# B&R Automation Studio project TrakDemo
Automation Studio 6.0.2.177; technology packages: mappCockpit 6.0.0, mappMotion 6.0.0, mappView 6.0.0, OpcUaCs 6.0.0

## Configuration Config1

CPU 5PC900.TS17-00, AutomationRuntime 6.0.2, Build 11.3.0, Safety 0.0, Vc 

### Task classes (Cpu.sw)
```
Cyclic#1:
  TrakInit <- Trak.TrakInit.prg
Cyclic#2:
  AssCtrl1 <- Trak.AssCtrl1.prg
  AssCtrl2 <- Trak.AssCtrl2.prg
DataObjects: McAcpSys
NcDataObjects: mcdrivelog
Binaries: FWRules, McAcpSim, arcoal, arsvcreg, TCData, McAcpDrv, mCoWebSc, mvLoader, arflatprv, udbdef, iomap, Config_1, arconfig, asfw, ashwac, sysconf, User, Settings, Role, ashwd, Config_4, Config_3, Config_2, Config, Hierarchy
Libraries: McBase, CoTrace, AsZip, FileIO, runtime, McAxis, McAcpTrak, MpBase, TrakLib, standard, AsBrStr, sys_lib, brsystem, TrakDiag, astime, ArEventLog, DataObj, AsHttp, AsArSdm, MpAxis, McAcpAx, powerlnk, arssl, asieccon, asepl
```

### Hardware
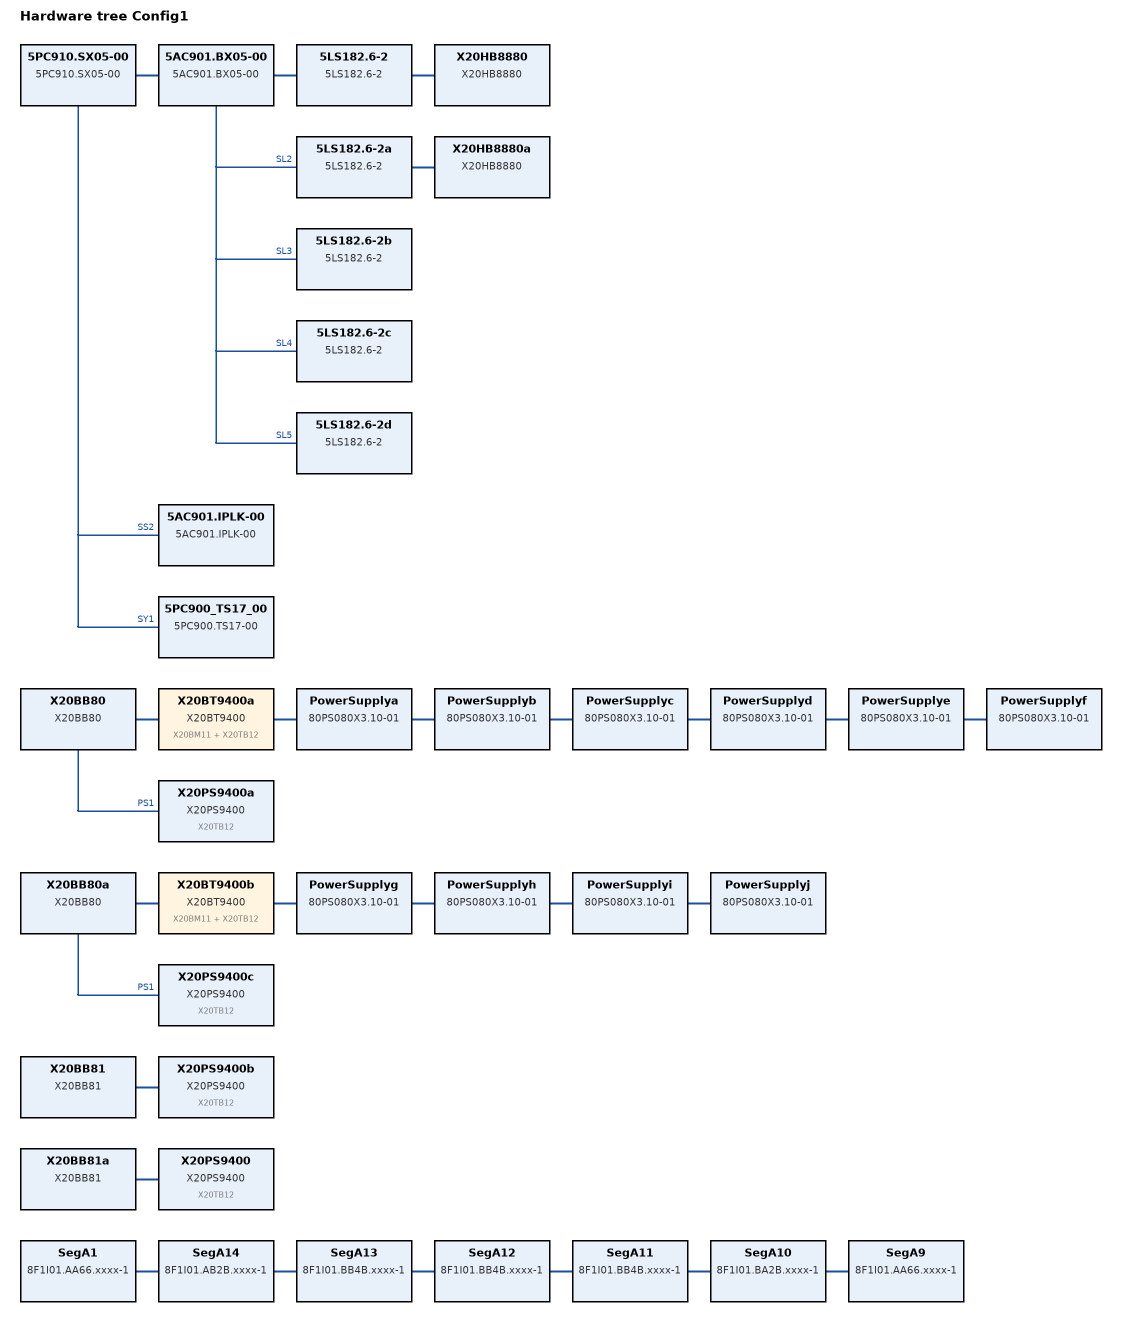
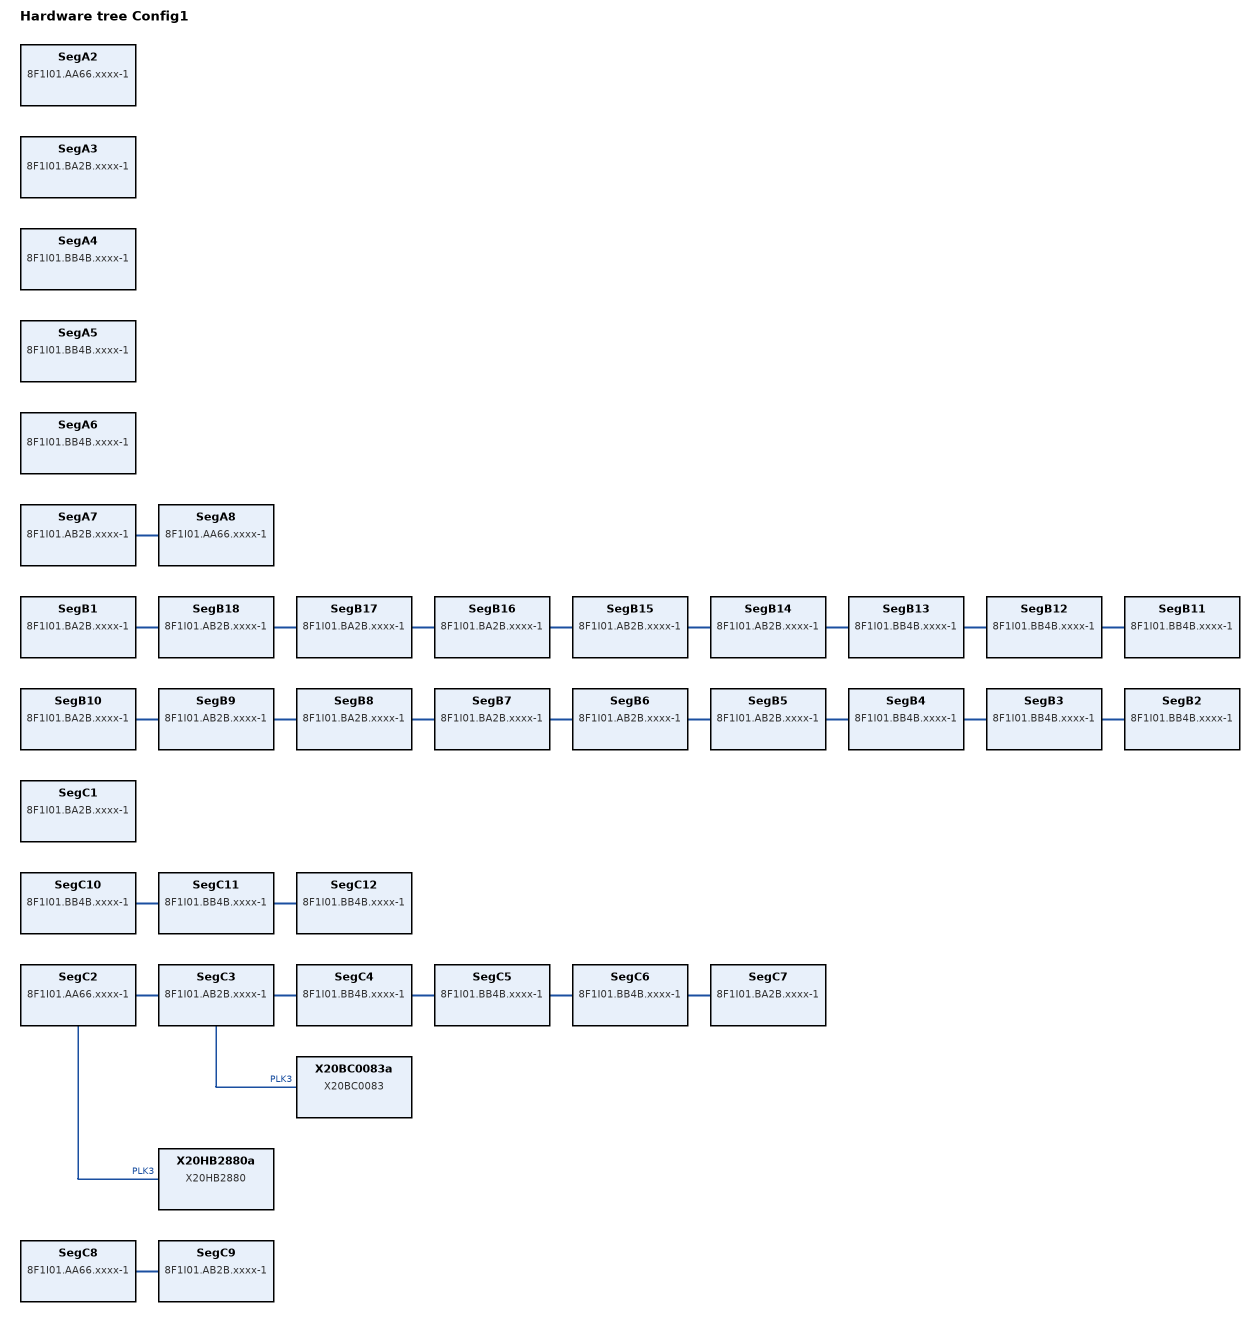
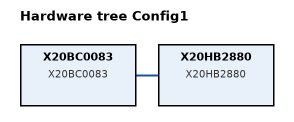
```
5AC901.BX05-00 : 5AC901.BX05-00 v1.0.1.0  [SY -> 5PC910.SX05-00.SY3]
5AC901.IPLK-00 : 5AC901.IPLK-00 v2.0.0.0 (Disabled=true)  [SS -> 5PC910.SX05-00.SS2]
  Connector IF1 (Disabled=true)
5LS182.6-2 : 5LS182.6-2 v1.12.0.0  [SL -> 5AC901.BX05-00.SL1]
  Connector IF1:
    NodeDefinition = Software
5LS182.6-2a : 5LS182.6-2 v1.12.0.0  [SL -> 5AC901.BX05-00.SL2]
5LS182.6-2b : 5LS182.6-2 v1.12.0.0 (Disabled=true)  [SL -> 5AC901.BX05-00.SL3]
  Connector IF1 (Disabled=true)
5LS182.6-2c : 5LS182.6-2 v1.12.0.0 (Disabled=true)  [SL -> 5AC901.BX05-00.SL4]
  Connector IF1 (Disabled=true)
5LS182.6-2d : 5LS182.6-2 v1.12.0.0 (Disabled=true)  [SL -> 5AC901.BX05-00.SL5]
  Connector IF1 (Disabled=true)
5PC900_TS17_00 : 5PC900.TS17-00 v2.1.0.0  [SY -> 5PC910.SX05-00.SY1]
  ConfigurationID = TrakDemo_Config1
  ConfigVersion = 1.2.3
  MotionLoggerSize = 2048000
  SystemTick = 2000
  TaskClassIdleTime = 10000
  Cyclic1Tolerance = 0
  FileDevice1
  FileDeviceName1 = SvgData
  FileDevicePath1 = USER_PATH\web\SvgData
  FileDevice2
  FileDeviceName2 = Diagnosis
  FileDevicePath2 = USER_PATH\web\Diagnosis
  EthernetDefaultGateway = 10.24.153.1
  ActivateFtpServer = 1
  FtpUser1
  FtpUsername1 = bur
  FtpUserPassword1 = efcpoAfz3gk2rn0a9Nq2v7CfehAGIZc7rIbAOhV34KU=
  FtpUserSalt1 = 5Q6RY3ay
  FTPAccessRight1 = 0
  ActivateWebServer = 1
  WebServerProtocol = 1
  WebServerWebDir = F:\web\
  ActivateSdm = 1
5PC910.SX05-00 : 5PC910.SX05-00 v2.1.2.0
  Connector IF1:
    AssignedOperatingSystem = ARemb
  Connector IF3:
    AssignedOperatingSystem = ARemb
    ActivateDevice = 1
    Mode = Manual
    InternetAddress = 10.24.153.43
    SubnetMask = 255.255.255.192
    ActivateIna = 0
    ActivateSnmp = 2
  Connector IF4:
    AssignedOperatingSystem = ARemb
    ActivateDevice = 1
  Connector IF5:
    AssignedOperatingSystem = ARemb
  Connector IF6:
    AssignedOperatingSystem = ARemb
  Connector IF7:
    AssignedOperatingSystem = ARemb
  Connector IF8:
    AssignedOperatingSystem = ARemb
  Connector IF9:
    AssignedOperatingSystem = ARemb
PowerSupplya : 80PS080X3.10-01 v1.7.0.0  [X2X1 -> X20BT9400a.X2X1 [Cable Type=X2XCable, Length=10, Version=1.0.0.3]]
  Supervision = off
PowerSupplyb : 80PS080X3.10-01 v1.7.0.0  [X2X1 -> PowerSupplya.X2X2 [Cable Type=X2XCable, Length=10, Version=1.0.0.3]]
  Supervision = off
PowerSupplyc : 80PS080X3.10-01 v1.7.0.0  [X2X1 -> PowerSupplyb.X2X2 [Cable Type=X2XCable, Length=10, Version=1.0.0.3]]
  Supervision = off
PowerSupplyd : 80PS080X3.10-01 v1.7.0.0  [X2X1 -> PowerSupplyc.X2X2 [Cable Type=X2XCable, Length=10, Version=1.0.0.3]]
  Supervision = off
PowerSupplye : 80PS080X3.10-01 v1.7.0.0  [X2X1 -> PowerSupplyd.X2X2 [Cable Type=X2XCable, Length=10, Version=1.0.0.3]]
  Supervision = off
PowerSupplyf : 80PS080X3.10-01 v1.7.0.0  [X2X1 -> PowerSupplye.X2X2 [Cable Type=X2XCable, Length=10, Version=1.0.0.3]]
  Supervision = off
PowerSupplyg : 80PS080X3.10-01 v1.7.0.0  [X2X1 -> X20BT9400b.X2X1 [Cable Type=X2XCable, Length=10, Version=1.0.0.3]]
  Supervision = off
PowerSupplyh : 80PS080X3.10-01 v1.7.0.0  [X2X1 -> PowerSupplyg.X2X2 [Cable Type=X2XCable, Length=10, Version=1.0.0.3]]
  Supervision = off
PowerSupplyi : 80PS080X3.10-01 v1.7.0.0  [X2X1 -> PowerSupplyh.X2X2 [Cable Type=X2XCable, Length=10, Version=1.0.0.3]]
  Supervision = off
PowerSupplyj : 80PS080X3.10-01 v1.7.0.0  [X2X1 -> PowerSupplyi.X2X2 [Cable Type=X2XCable, Length=10, Version=1.0.0.3]]
  Supervision = off
SegA1 : 8F1I01.AA66.xxxx-1 v1.0.0.4 (NodeNumber=1)  [PLK1 -> SegA2.PLK2 [Cable Type=PowerlinkCable, Length=10, Version=1.0.0.3]; PLK2 -> SegA14.PLK1 [Cable Type=PowerlinkCable, Length=10, Version=1.0.0.3]; PLK3 -> X20HB8880.ETH2 [Cable Type=PowerlinkCable, Length=10, Version=1.0.0.3]]
  DriveConfiguration:
    McTypeID = LLMConfig
  DriveConfiguration/Segment:
    Shape = STRAIGHT660
    SegmentReference = gSegA1
    SegmentSectorDirection = Positive
    ElongationCompensation = UseAssemblySetting
    StopReaction = UseAssemblySetting
    SpeedFilter = UseAssemblySetting
SegA10 : 8F1I01.BA2B.xxxx-1 v1.0.0.4 (NodeNumber=25)  [PLK1 -> SegA11.PLK2 [Cable Type=PowerlinkCable, Length=10, Version=1.0.0.3]; PLK2 -> SegA9.PLK1 [Cable Type=PowerlinkCable, Length=10, Version=1.0.0.3]]
  DriveConfiguration:
    McTypeID = LLMConfig
  DriveConfiguration/Segment:
    Shape = CIRCULAR_TO_STRAIGHT105
    SegmentReference = gSegA10
    SegmentSectorDirection = Positive
    ElongationCompensation = UseAssemblySetting
    StopReaction = UseAssemblySetting
    SpeedFilter = UseAssemblySetting
SegA11 : 8F1I01.BB4B.xxxx-1 v1.0.0.4 (NodeNumber=24)  [PLK1 -> SegA12.PLK2 [Cable Type=PowerlinkCable, Length=10, Version=1.0.0.3]; PLK2 -> SegA10.PLK1 [Cable Type=PowerlinkCable, Length=10, Version=1.0.0.3]]
  DriveConfiguration:
    McTypeID = LLMConfig
  DriveConfiguration/Segment:
    Shape = CIRCULAR
    SegmentReference = gSegA11
    SegmentSectorDirection = Positive
    ElongationCompensation = UseAssemblySetting
    StopReaction = UseAssemblySetting
    SpeedFilter = UseAssemblySetting
SegA12 : 8F1I01.BB4B.xxxx-1 v1.0.0.4 (NodeNumber=23)  [PLK1 -> SegA13.PLK2 [Cable Type=PowerlinkCable, Length=10, Version=1.0.0.3]; PLK2 -> SegA11.PLK1 [Cable Type=PowerlinkCable, Length=10, Version=1.0.0.3]]
  DriveConfiguration:
    McTypeID = LLMConfig
  DriveConfiguration/Segment:
    Shape = CIRCULAR
    SegmentReference = gSegA12
    SegmentSectorDirection = Positive
    ElongationCompensation = UseAssemblySetting
    StopReaction = UseAssemblySetting
    SpeedFilter = UseAssemblySetting
SegA13 : 8F1I01.BB4B.xxxx-1 v1.0.0.4 (NodeNumber=22)  [PLK1 -> SegA14.PLK2 [Cable Type=PowerlinkCable, Length=10, Version=1.0.0.3]; PLK2 -> SegA12.PLK1 [Cable Type=PowerlinkCable, Length=10, Version=1.0.0.3]]
  DriveConfiguration:
    McTypeID = LLMConfig
  DriveConfiguration/Segment:
    Shape = CIRCULAR
    SegmentReference = gSegA13
    SegmentSectorDirection = Positive
    ElongationCompensation = UseAssemblySetting
    StopReaction = UseAssemblySetting
    SpeedFilter = UseAssemblySetting
SegA14 : 8F1I01.AB2B.xxxx-1 v1.0.0.4 (NodeNumber=21)  [PLK1 -> SegA1.PLK2 [Cable Type=PowerlinkCable, Length=10, Version=1.0.0.3]; PLK2 -> SegA13.PLK1 [Cable Type=PowerlinkCable, Length=10, Version=1.0.0.3]]
  DriveConfiguration:
    McTypeID = LLMConfig
  DriveConfiguration/Segment:
    Shape = STRAIGHT105_TO_CIRCULAR
    SegmentReference = gSegA14
    SegmentSectorDirection = Positive
    ElongationCompensation = UseAssemblySetting
    StopReaction = UseAssemblySetting
    SpeedFilter = UseAssemblySetting
SegA2 : 8F1I01.AA66.xxxx-1 v1.0.0.4 (NodeNumber=2)  [PLK1 -> SegA3.PLK2 [Cable Type=PowerlinkCable, Length=10, Version=1.0.0.3]; PLK2 -> SegA1.PLK1 [Cable Type=PowerlinkCable, Length=10, Version=1.0.0.3]]
  DriveConfiguration:
    McTypeID = LLMConfig
  DriveConfiguration/Segment:
    Shape = STRAIGHT660
    SegmentReference = gSegA2
    SegmentSectorDirection = Positive
    ElongationCompensation = UseAssemblySetting
    StopReaction = UseAssemblySetting
    SpeedFilter = UseAssemblySetting
SegA3 : 8F1I01.BA2B.xxxx-1 v1.0.0.4 (NodeNumber=27)  [PLK1 -> SegA4.PLK2 [Cable Type=PowerlinkCable, Length=10, Version=1.0.0.3]; PLK2 -> SegA2.PLK1 [Cable Type=PowerlinkCable, Length=10, Version=1.0.0.3]]
  DriveConfiguration:
    McTypeID = LLMConfig
  DriveConfiguration/Segment:
    Shape = CIRCULAR_TO_STRAIGHT105
    SegmentReference = gSegA3
    SegmentSectorDirection = Positive
    ElongationCompensation = UseAssemblySetting
    StopReaction = UseAssemblySetting
    SpeedFilter = UseAssemblySetting
SegA4 : 8F1I01.BB4B.xxxx-1 v1.0.0.4 (NodeNumber=28)  [PLK1 -> SegA5.PLK2 [Cable Type=PowerlinkCable, Length=10, Version=1.0.0.3]; PLK2 -> SegA3.PLK1 [Cable Type=PowerlinkCable, Length=10, Version=1.0.0.3]]
  DriveConfiguration:
    McTypeID = LLMConfig
  DriveConfiguration/Segment:
    Shape = CIRCULAR
    SegmentReference = gSegA4
    SegmentSectorDirection = Positive
    ElongationCompensation = UseAssemblySetting
    StopReaction = UseAssemblySetting
    SpeedFilter = UseAssemblySetting
SegA5 : 8F1I01.BB4B.xxxx-1 v1.0.0.4 (NodeNumber=29)  [PLK1 -> SegA6.PLK2 [Cable Type=PowerlinkCable, Length=10, Version=1.0.0.3]; PLK2 -> SegA4.PLK1 [Cable Type=PowerlinkCable, Length=10, Version=1.0.0.3]]
  DriveConfiguration:
    McTypeID = LLMConfig
  DriveConfiguration/Segment:
    Shape = CIRCULAR
    SegmentReference = gSegA5
    SegmentSectorDirection = Positive
    ElongationCompensation = UseAssemblySetting
    StopReaction = UseAssemblySetting
    SpeedFilter = UseAssemblySetting
SegA6 : 8F1I01.BB4B.xxxx-1 v1.0.0.4 (NodeNumber=30)  [PLK1 -> SegA7.PLK2 [Cable Type=PowerlinkCable, Length=10, Version=1.0.0.3]; PLK2 -> SegA5.PLK1 [Cable Type=PowerlinkCable, Length=10, Version=1.0.0.3]]
  DriveConfiguration:
    McTypeID = LLMConfig
  DriveConfiguration/Segment:
    Shape = CIRCULAR
    SegmentReference = gSegA6
    SegmentSectorDirection = Positive
    ElongationCompensation = UseAssemblySetting
    StopReaction = UseAssemblySetting
    SpeedFilter = UseAssemblySetting
SegA7 : 8F1I01.AB2B.xxxx-1 v1.0.0.4 (NodeNumber=31)  [PLK1 -> SegA8.PLK2 [Cable Type=PowerlinkCable, Length=10, Version=1.0.0.3]; PLK2 -> SegA6.PLK1 [Cable Type=PowerlinkCable, Length=10, Version=1.0.0.3]]
  DriveConfiguration:
    McTypeID = LLMConfig
  DriveConfiguration/Segment:
    Shape = STRAIGHT105_TO_CIRCULAR
    SegmentReference = gSegA7
    SegmentSectorDirection = Positive
    ElongationCompensation = UseAssemblySetting
    StopReaction = UseAssemblySetting
    SpeedFilter = UseAssemblySetting
SegA8 : 8F1I01.AA66.xxxx-1 v1.0.0.4 (NodeNumber=32)  [PLK2 -> SegA7.PLK1 [Cable Type=PowerlinkCable, Length=10, Version=1.0.0.3]]
  DriveConfiguration:
    McTypeID = LLMConfig
  DriveConfiguration/Segment:
    Shape = STRAIGHT660
    SegmentReference = gSegA8
    SegmentSectorDirection = Positive
    ElongationCompensation = UseAssemblySetting
    StopReaction = UseAssemblySetting
    SpeedFilter = UseAssemblySetting
SegA9 : 8F1I01.AA66.xxxx-1 v1.0.0.4 (NodeNumber=26)  [PLK1 -> SegA10.PLK2 [Cable Type=PowerlinkCable, Length=10, Version=1.0.0.3]]
  DriveConfiguration:
    McTypeID = LLMConfig
  DriveConfiguration/Segment:
    Shape = STRAIGHT660
    SegmentReference = gSegA9
    SegmentSectorDirection = Positive
    ElongationCompensation = UseAssemblySetting
    StopReaction = UseAssemblySetting
    SpeedFilter = UseAssemblySetting
SegB1 : 8F1I01.BA2B.xxxx-1 v1.0.0.4 (NodeNumber=3)  [PLK1 -> SegB2.PLK2 [Cable Type=PowerlinkCable, Length=10, Version=1.0.0.3]; PLK2 -> SegB18.PLK1 [Cable Type=PowerlinkCable, Length=10, Version=1.0.0.3]; PLK3 -> X20HB2880.ETH2 [Cable Type=PowerlinkCable, Length=10, Version=1.0.0.3]]
  DriveConfiguration:
    McTypeID = LLMConfig
  DriveConfiguration/Segment:
    Shape = CIRCULAR_TO_STRAIGHT105
    SegmentReference = gSegB1
    SegmentSectorDirection = Positive
    ElongationCompensation = UseAssemblySetting
    StopReaction = UseAssemblySetting
    SpeedFilter = UseAssemblySetting
SegB10 : 8F1I01.BA2B.xxxx-1 v1.0.0.4 (NodeNumber=12)  [PLK2 -> SegB9.PLK1 [Cable Type=PowerlinkCable, Length=10, Version=1.0.0.3]]
  DriveConfiguration:
    McTypeID = LLMConfig
  DriveConfiguration/Segment:
    Shape = CIRCULAR_TO_STRAIGHT105
    SegmentReference = gSegB10
    SegmentSectorDirection = Positive
    ElongationCompensation = UseAssemblySetting
    StopReaction = UseAssemblySetting
    SpeedFilter = UseAssemblySetting
SegB11 : 8F1I01.BB4B.xxxx-1 v1.0.0.4 (NodeNumber=11)  [PLK1 -> SegB12.PLK2 [Cable Type=PowerlinkCable, Length=10, Version=1.0.0.3]]
  DriveConfiguration:
    McTypeID = LLMConfig
  DriveConfiguration/Segment:
    Shape = CIRCULAR
    SegmentReference = gSegB11
    SegmentSectorDirection = Positive
    ElongationCompensation = UseAssemblySetting
    StopReaction = UseAssemblySetting
    SpeedFilter = UseAssemblySetting
SegB12 : 8F1I01.BB4B.xxxx-1 v1.0.0.4 (NodeNumber=10)  [PLK1 -> SegB13.PLK2 [Cable Type=PowerlinkCable, Length=10, Version=1.0.0.3]; PLK2 -> SegB11.PLK1 [Cable Type=PowerlinkCable, Length=10, Version=1.0.0.3]]
  DriveConfiguration:
    McTypeID = LLMConfig
  DriveConfiguration/Segment:
    Shape = CIRCULAR
    SegmentReference = gSegB12
    SegmentSectorDirection = Positive
    ElongationCompensation = UseAssemblySetting
    StopReaction = UseAssemblySetting
    SpeedFilter = UseAssemblySetting
SegB13 : 8F1I01.BB4B.xxxx-1 v1.0.0.4 (NodeNumber=9)  [PLK1 -> SegB14.PLK2 [Cable Type=PowerlinkCable, Length=10, Version=1.0.0.3]; PLK2 -> SegB12.PLK1 [Cable Type=PowerlinkCable, Length=10, Version=1.0.0.3]]
  DriveConfiguration:
    McTypeID = LLMConfig
  DriveConfiguration/Segment:
    Shape = CIRCULAR
    SegmentReference = gSegB13
    SegmentSectorDirection = Positive
    ElongationCompensation = UseAssemblySetting
    StopReaction = UseAssemblySetting
    SpeedFilter = UseAssemblySetting
SegB14 : 8F1I01.AB2B.xxxx-1 v1.0.0.4 (NodeNumber=8)  [PLK1 -> SegB15.PLK2 [Cable Type=PowerlinkCable, Length=10, Version=1.0.0.3]; PLK2 -> SegB13.PLK1 [Cable Type=PowerlinkCable, Length=10, Version=1.0.0.3]]
  DriveConfiguration:
    McTypeID = LLMConfig
  DriveConfiguration/Segment:
    Shape = STRAIGHT105_TO_CIRCULAR
    SegmentReference = gSegB14
    SegmentSectorDirection = Positive
    ElongationCompensation = UseAssemblySetting
    StopReaction = UseAssemblySetting
    SpeedFilter = UseAssemblySetting
SegB15 : 8F1I01.AB2B.xxxx-1 v1.0.0.4 (NodeNumber=7)  [PLK1 -> SegB16.PLK2 [Cable Type=PowerlinkCable, Length=10, Version=1.0.0.3]; PLK2 -> SegB14.PLK1 [Cable Type=PowerlinkCable, Length=10, Version=1.0.0.3]]
  DriveConfiguration:
    McTypeID = LLMConfig
  DriveConfiguration/Segment:
    Shape = STRAIGHT105_TO_CIRCULAR
    SegmentReference = gSegB15
    SegmentSectorDirection = Positive
    ElongationCompensation = UseAssemblySetting
    StopReaction = UseAssemblySetting
    SpeedFilter = UseAssemblySetting
SegB16 : 8F1I01.BA2B.xxxx-1 v1.0.0.4 (NodeNumber=6)  [PLK1 -> SegB17.PLK2 [Cable Type=PowerlinkCable, Length=10, Version=1.0.0.3]; PLK2 -> SegB15.PLK1 [Cable Type=PowerlinkCable, Length=10, Version=1.0.0.3]]
  DriveConfiguration:
    McTypeID = LLMConfig
  DriveConfiguration/Segment:
    Shape = CIRCULAR_TO_STRAIGHT105
    SegmentReference = gSegB16
    SegmentSectorDirection = Positive
    ElongationCompensation = UseAssemblySetting
    StopReaction = UseAssemblySetting
    SpeedFilter = UseAssemblySetting
SegB17 : 8F1I01.BA2B.xxxx-1 v1.0.0.4 (NodeNumber=5)  [PLK1 -> SegB18.PLK2 [Cable Type=PowerlinkCable, Length=10, Version=1.0.0.3]; PLK2 -> SegB16.PLK1 [Cable Type=PowerlinkCable, Length=10, Version=1.0.0.3]]
  DriveConfiguration:
    McTypeID = LLMConfig
  DriveConfiguration/Segment:
    Shape = CIRCULAR_TO_STRAIGHT105
    SegmentReference = gSegB17
    SegmentSectorDirection = Positive
    ElongationCompensation = UseAssemblySetting
    StopReaction = UseAssemblySetting
    SpeedFilter = UseAssemblySetting
SegB18 : 8F1I01.AB2B.xxxx-1 v1.0.0.4 (NodeNumber=4)  [PLK1 -> SegB1.PLK2 [Cable Type=PowerlinkCable, Length=10, Version=1.0.0.3]; PLK2 -> SegB17.PLK1 [Cable Type=PowerlinkCable, Length=10, Version=1.0.0.3]]
  DriveConfiguration:
    McTypeID = LLMConfig
  DriveConfiguration/Segment:
    Shape = STRAIGHT105_TO_CIRCULAR
    SegmentReference = gSegB18
    SegmentSectorDirection = Positive
    ElongationCompensation = UseAssemblySetting
    StopReaction = UseAssemblySetting
    SpeedFilter = UseAssemblySetting
SegB2 : 8F1I01.BB4B.xxxx-1 v1.0.0.4 (NodeNumber=13)  [PLK1 -> SegB3.PLK2 [Cable Type=PowerlinkCable, Length=10, Version=1.0.0.3]; PLK2 -> SegB1.PLK1 [Cable Type=PowerlinkCable, Length=10, Version=1.0.0.3]]
  DriveConfiguration:
    McTypeID = LLMConfig
  DriveConfiguration/Segment:
    Shape = CIRCULAR
    SegmentReference = gSegB2
    SegmentSectorDirection = Positive
    ElongationCompensation = UseAssemblySetting
    StopReaction = UseAssemblySetting
    SpeedFilter = UseAssemblySetting
SegB3 : 8F1I01.BB4B.xxxx-1 v1.0.0.4 (NodeNumber=14)  [PLK1 -> SegB4.PLK2 [Cable Type=PowerlinkCable, Length=10, Version=1.0.0.3]; PLK2 -> SegB2.PLK1 [Cable Type=PowerlinkCable, Length=10, Version=1.0.0.3]]
  DriveConfiguration:
    McTypeID = LLMConfig
  DriveConfiguration/Segment:
    Shape = CIRCULAR
    SegmentReference = gSegB3
    SegmentSectorDirection = Positive
    ElongationCompensation = UseAssemblySetting
    StopReaction = UseAssemblySetting
    SpeedFilter = UseAssemblySetting
SegB4 : 8F1I01.BB4B.xxxx-1 v1.0.0.4 (NodeNumber=15)  [PLK1 -> SegB5.PLK2 [Cable Type=PowerlinkCable, Length=10, Version=1.0.0.3]; PLK2 -> SegB3.PLK1 [Cable Type=PowerlinkCable, Length=10, Version=1.0.0.3]]
  DriveConfiguration:
    McTypeID = LLMConfig
  DriveConfiguration/Segment:
    Shape = CIRCULAR
    SegmentReference = gSegB4
    SegmentSectorDirection = Positive
    ElongationCompensation = UseAssemblySetting
    StopReaction = UseAssemblySetting
    SpeedFilter = UseAssemblySetting
SegB5 : 8F1I01.AB2B.xxxx-1 v1.0.0.4 (NodeNumber=16)  [PLK1 -> SegB6.PLK2 [Cable Type=PowerlinkCable, Length=10, Version=1.0.0.3]; PLK2 -> SegB4.PLK1 [Cable Type=PowerlinkCable, Length=10, Version=1.0.0.3]]
  DriveConfiguration:
    McTypeID = LLMConfig
  DriveConfiguration/Segment:
    Shape = STRAIGHT105_TO_CIRCULAR
    SegmentReference = gSegB5
    SegmentSectorDirection = Positive
    ElongationCompensation = UseAssemblySetting
    StopReaction = UseAssemblySetting
    SpeedFilter = UseAssemblySetting
SegB6 : 8F1I01.AB2B.xxxx-1 v1.0.0.4 (NodeNumber=17)  [PLK1 -> SegB7.PLK2 [Cable Type=PowerlinkCable, Length=10, Version=1.0.0.3]; PLK2 -> SegB5.PLK1 [Cable Type=PowerlinkCable, Length=10, Version=1.0.0.3]]
  DriveConfiguration:
    McTypeID = LLMConfig
  DriveConfiguration/Segment:
    Shape = STRAIGHT105_TO_CIRCULAR
    SegmentReference = gSegB6
    SegmentSectorDirection = Positive
    ElongationCompensation = UseAssemblySetting
    StopReaction = UseAssemblySetting
    SpeedFilter = UseAssemblySetting
SegB7 : 8F1I01.BA2B.xxxx-1 v1.0.0.4 (NodeNumber=18)  [PLK1 -> SegB8.PLK2 [Cable Type=PowerlinkCable, Length=10, Version=1.0.0.3]; PLK2 -> SegB6.PLK1 [Cable Type=PowerlinkCable, Length=10, Version=1.0.0.3]]
  DriveConfiguration:
    McTypeID = LLMConfig
  DriveConfiguration/Segment:
    Shape = CIRCULAR_TO_STRAIGHT105
    SegmentReference = gSegB7
    SegmentSectorReference = gSecB7
    SegmentSectorDirection = Positive
    ElongationCompensation = UseAssemblySetting
    ACC = Inactive
    StopReaction = UseAssemblySetting
    SpeedFilter = UseAssemblySetting
    PositionControllerLagMonitor = UseAssemblySetting
SegB8 : 8F1I01.BA2B.xxxx-1 v1.0.0.4 (NodeNumber=20)  [PLK1 -> SegB9.PLK2 [Cable Type=PowerlinkCable, Length=10, Version=1.0.0.3]; PLK2 -> SegB7.PLK1 [Cable Type=PowerlinkCable, Length=10, Version=1.0.0.3]]
  DriveConfiguration:
    McTypeID = LLMConfig
  DriveConfiguration/Segment:
    Shape = CIRCULAR_TO_STRAIGHT105
    SegmentReference = gSegB8
    SegmentSectorDirection = Positive
    ElongationCompensation = UseAssemblySetting
    StopReaction = UseAssemblySetting
    SpeedFilter = UseAssemblySetting
SegB9 : 8F1I01.AB2B.xxxx-1 v1.0.0.4 (NodeNumber=19)  [PLK1 -> SegB10.PLK2 [Cable Type=PowerlinkCable, Length=10, Version=1.0.0.3]; PLK2 -> SegB8.PLK1 [Cable Type=PowerlinkCable, Length=10, Version=1.0.0.3]]
  DriveConfiguration:
    McTypeID = LLMConfig
  DriveConfiguration/Segment:
    Shape = STRAIGHT105_TO_CIRCULAR
    SegmentReference = gSegB9
    SegmentSectorDirection = Positive
    ElongationCompensation = UseAssemblySetting
    StopReaction = UseAssemblySetting
    SpeedFilter = UseAssemblySetting
SegC1 : 8F1I01.BA2B.xxxx-1 v1.0.0.4 (NodeNumber=1)  [PLK1 -> SegC12.PLK2 [Cable Type=PowerlinkCable, Length=10, Version=1.0.0.3]; PLK3 -> X20HB8880a.ETH2 [Cable Type=PowerlinkCable, Length=10, Version=1.0.0.3]]
  DriveConfiguration:
    McTypeID = LLMConfig
  DriveConfiguration/Segment:
    Shape = CIRCULAR_TO_STRAIGHT105
    SegmentReference = gSegC1
    SegmentSectorReference = gSecC1
    SegmentSectorDirection = Positive
    ElongationCompensation = UseAssemblySetting
    ACC = Inactive
    StopReaction = UseAssemblySetting
    SpeedFilter = UseAssemblySetting
    PositionControllerLagMonitor = UseAssemblySetting
SegC10 : 8F1I01.BB4B.xxxx-1 v1.0.0.4  [PLK1 -> SegC9.PLK2 [Cable Type=PowerlinkCable, Length=10, Version=1.0.0.3]; PLK2 -> SegC11.PLK1 [Cable Type=PowerlinkCable, Length=10, Version=1.0.0.3]]
  DriveConfiguration:
    McTypeID = LLMConfig
  DriveConfiguration/Segment:
    Shape = CIRCULAR
    SegmentReference = gSegC10
    SegmentSectorDirection = Positive
    ElongationCompensation = UseAssemblySetting
    ACC = Inactive
    StopReaction = UseAssemblySetting
    SpeedFilter = UseAssemblySetting
    PositionControllerLagMonitor = UseAssemblySetting
SegC11 : 8F1I01.BB4B.xxxx-1 v1.0.0.4  [PLK1 -> SegC10.PLK2 [Cable Type=PowerlinkCable, Length=10, Version=1.0.0.3]; PLK2 -> SegC12.PLK1 [Cable Type=PowerlinkCable, Length=10, Version=1.0.0.3]]
  DriveConfiguration:
    McTypeID = LLMConfig
  DriveConfiguration/Segment:
    Shape = CIRCULAR
    SegmentReference = gSegC11
    SegmentSectorDirection = Positive
    ElongationCompensation = UseAssemblySetting
    ACC = Inactive
    StopReaction = UseAssemblySetting
    SpeedFilter = UseAssemblySetting
    PositionControllerLagMonitor = UseAssemblySetting
SegC12 : 8F1I01.BB4B.xxxx-1 v1.0.0.4 (NodeNumber=3)  [PLK1 -> SegC11.PLK2 [Cable Type=PowerlinkCable, Length=10, Version=1.0.0.3]; PLK2 -> SegC1.PLK1 [Cable Type=PowerlinkCable, Length=10, Version=1.0.0.3]]
  DriveConfiguration:
    McTypeID = LLMConfig
  DriveConfiguration/Segment:
    Shape = CIRCULAR
    SegmentReference = gSegC12
    SegmentSectorDirection = Positive
    ElongationCompensation = UseAssemblySetting
    ACC = Inactive
    StopReaction = UseAssemblySetting
    SpeedFilter = UseAssemblySetting
    PositionControllerLagMonitor = UseAssemblySetting
SegC2 : 8F1I01.AA66.xxxx-1 v1.0.0.4 (NodeNumber=2)  [PLK2 -> SegC3.PLK1 [Cable Type=PowerlinkCable, Length=10, Version=1.0.0.3]; PLK3 -> X20HB2880a.ETH2 [Cable Type=PowerlinkCable, Length=10, Version=1.0.0.3]]
  DriveConfiguration:
    McTypeID = LLMConfig
  DriveConfiguration/Segment:
    Shape = STRAIGHT660
    SegmentReference = gSegC2
    SegmentSectorDirection = Positive
    ElongationCompensation = UseAssemblySetting
    ACC = Inactive
    StopReaction = UseAssemblySetting
    SpeedFilter = UseAssemblySetting
    PositionControllerLagMonitor = UseAssemblySetting
SegC3 : 8F1I01.AB2B.xxxx-1 v1.0.0.4 (NodeNumber=12)  [PLK1 -> SegC2.PLK2 [Cable Type=PowerlinkCable, Length=10, Version=1.0.0.3]; PLK2 -> SegC4.PLK1 [Cable Type=PowerlinkCable, Length=10, Version=1.0.0.3]; PLK3 -> X20BC0083a.PLK1 [Cable Type=PowerlinkCable, Length=10, Version=1.0.0.3]]
  DriveConfiguration:
    McTypeID = LLMConfig
  DriveConfiguration/Segment:
    Shape = STRAIGHT105_TO_CIRCULAR
    SegmentReference = gSegC3
    SegmentSectorDirection = Positive
    ElongationCompensation = UseAssemblySetting
    ACC = Inactive
    StopReaction = UseAssemblySetting
    SpeedFilter = UseAssemblySetting
    PositionControllerLagMonitor = UseAssemblySetting
SegC4 : 8F1I01.BB4B.xxxx-1 v1.0.0.4 (NodeNumber=11)  [PLK1 -> SegC3.PLK2 [Cable Type=PowerlinkCable, Length=10, Version=1.0.0.3]; PLK2 -> SegC5.PLK1 [Cable Type=PowerlinkCable, Length=10, Version=1.0.0.3]]
  DriveConfiguration:
    McTypeID = LLMConfig
  DriveConfiguration/Segment:
    Shape = CIRCULAR
    SegmentReference = gSegC4
    SegmentSectorDirection = Positive
    ElongationCompensation = UseAssemblySetting
    ACC = Inactive
    StopReaction = UseAssemblySetting
    SpeedFilter = UseAssemblySetting
    PositionControllerLagMonitor = UseAssemblySetting
SegC5 : 8F1I01.BB4B.xxxx-1 v1.0.0.4 (NodeNumber=10)  [PLK1 -> SegC4.PLK2 [Cable Type=PowerlinkCable, Length=10, Version=1.0.0.3]; PLK2 -> SegC6.PLK1 [Cable Type=PowerlinkCable, Length=10, Version=1.0.0.3]]
  DriveConfiguration:
    McTypeID = LLMConfig
  DriveConfiguration/Segment:
    Shape = CIRCULAR
    SegmentReference = gSegC5
    SegmentSectorDirection = Positive
    ElongationCompensation = UseAssemblySetting
    ACC = Inactive
    StopReaction = UseAssemblySetting
    SpeedFilter = UseAssemblySetting
    PositionControllerLagMonitor = UseAssemblySetting
SegC6 : 8F1I01.BB4B.xxxx-1 v1.0.0.4 (NodeNumber=9)  [PLK1 -> SegC5.PLK2 [Cable Type=PowerlinkCable, Length=10, Version=1.0.0.3]; PLK2 -> SegC7.PLK1 [Cable Type=PowerlinkCable, Length=10, Version=1.0.0.3]]
  DriveConfiguration:
    McTypeID = LLMConfig
  DriveConfiguration/Segment:
    Shape = CIRCULAR
    SegmentReference = gSegC6
    SegmentSectorDirection = Positive
    ElongationCompensation = UseAssemblySetting
    ACC = Inactive
    StopReaction = UseAssemblySetting
    SpeedFilter = UseAssemblySetting
    PositionControllerLagMonitor = UseAssemblySetting
SegC7 : 8F1I01.BA2B.xxxx-1 v1.0.0.4 (NodeNumber=8)  [PLK1 -> SegC6.PLK2 [Cable Type=PowerlinkCable, Length=10, Version=1.0.0.3]]
  DriveConfiguration:
    McTypeID = LLMConfig
  DriveConfiguration/Segment:
    Shape = CIRCULAR_TO_STRAIGHT105
    SegmentReference = gSegC7
    SegmentSectorReference = gSecC7
    SegmentSectorDirection = Positive
    ElongationCompensation = UseAssemblySetting
    ACC = Inactive
    StopReaction = UseAssemblySetting
    SpeedFilter = UseAssemblySetting
    PositionControllerLagMonitor = UseAssemblySetting
SegC8 : 8F1I01.AA66.xxxx-1 v1.0.0.4 (NodeNumber=7)  [PLK2 -> SegC9.PLK1 [Cable Type=PowerlinkCable, Length=10, Version=1.0.0.3]]
  DriveConfiguration:
    McTypeID = LLMConfig
  DriveConfiguration/Segment:
    Shape = STRAIGHT660
    SegmentReference = gSegC8
    SegmentSectorDirection = Positive
    ElongationCompensation = UseAssemblySetting
    ACC = Inactive
    StopReaction = UseAssemblySetting
    SpeedFilter = UseAssemblySetting
    PositionControllerLagMonitor = UseAssemblySetting
SegC9 : 8F1I01.AB2B.xxxx-1 v1.0.0.4 (NodeNumber=6)  [PLK1 -> SegC8.PLK2 [Cable Type=PowerlinkCable, Length=10, Version=1.0.0.3]; PLK2 -> SegC10.PLK1 [Cable Type=PowerlinkCable, Length=10, Version=1.0.0.3]]
  DriveConfiguration:
    McTypeID = LLMConfig
  DriveConfiguration/Segment:
    Shape = STRAIGHT105_TO_CIRCULAR
    SegmentReference = gSegC9
    SegmentSectorDirection = Positive
    ElongationCompensation = UseAssemblySetting
    ACC = Inactive
    StopReaction = UseAssemblySetting
    SpeedFilter = UseAssemblySetting
    PositionControllerLagMonitor = UseAssemblySetting
X20BB80 : X20BB80 v1.1.0.0
X20BB80a : X20BB80 v1.1.0.0
X20BB81 : X20BB81 v1.2.0.0
  Connector IF1:
    ActivateX2X = 0
X20BB81a : X20BB81 v1.2.0.0
  Connector IF1:
    ActivateX2X = 0
X20BC0083 : X20BC0083 v2.16.1.0 (NodeNumber=33)  [PLK1 -> X20HB2880.ETH1 [Cable Type=PowerlinkCable, Length=10, Version=1.0.0.3]; SL -> X20BB80.SL1]
  Supervision = off
X20BC0083a : X20BC0083 v2.16.1.0 (NodeNumber=33)  [PLK1 -> SegC3.PLK3 [Cable Type=PowerlinkCable, Length=10, Version=1.0.0.3]; SL -> X20BB80a.SL1]
  Supervision = off
X20BM11 : X20BM11 v1.1.0.0  [X2X1 -> X20BB80.IF1]
X20BM11a : X20BM11 v1.1.0.0  [X2X1 -> X20BB80a.IF1]
X20BT9400a : X20BT9400 v1.3.1.0  [SS1 -> X20TB12b.SS; SL -> X20BM11.SL1]
  Supervision = off
X20BT9400b : X20BT9400 v1.3.1.0  [SS1 -> X20TB12e.SS; SL -> X20BM11a.SL1]
  Supervision = off
X20HB2880 : X20HB2880 v1.2.1.0  [ETH1 -> X20BC0083.PLK1 [Cable Type=PowerlinkCable, Length=10, Version=1.0.0.3]; ETH2 -> SegB1.PLK3 [Cable Type=PowerlinkCable, Length=10, Version=1.0.0.3]; SS -> X20BB81a.SS1]
X20HB2880a : X20HB2880 v1.2.1.0  [ETH2 -> SegC2.PLK3 [Cable Type=PowerlinkCable, Length=10, Version=1.0.0.3]; SS -> X20BB81.SS1]
X20HB8880 : X20HB8880 v1.1.1.0  [ETH1 -> 5LS182.6-2.IF1 [Cable Type=PowerlinkCable, Length=10, Version=1.0.0.3]; ETH2 -> SegA1.PLK3 [Cable Type=PowerlinkCable, Length=10, Version=1.0.0.3]; SL -> X20BB81a.SL1]
X20HB8880a : X20HB8880 v1.1.1.0  [ETH1 -> 5LS182.6-2a.IF1 [Cable Type=PowerlinkCable, Length=10, Version=1.0.0.3]; ETH2 -> SegC1.PLK3 [Cable Type=PowerlinkCable, Length=10, Version=1.0.0.3]; SL -> X20BB81.SL1]
X20PS9400 : X20PS9400 v1.8.1.0  [SS1 -> X20TB12.SS; PS -> X20BB81a.PS1]
  Supervision = off
X20PS9400a : X20PS9400 v1.8.1.0  [SS1 -> X20TB12a.SS; PS -> X20BB80.PS1]
  Supervision = off
X20PS9400b : X20PS9400 v1.8.1.0  [SS1 -> X20TB12c.SS; PS -> X20BB81.PS1]
  Supervision = off
X20PS9400c : X20PS9400 v1.8.1.0  [SS1 -> X20TB12d.SS; PS -> X20BB80a.PS1]
  Supervision = off
X20TB12 : X20TB12 v1.0.0.0
X20TB12a : X20TB12 v1.0.0.0
X20TB12b : X20TB12 v1.0.0.0
X20TB12c : X20TB12 v1.0.0.0
X20TB12d : X20TB12 v1.0.0.0
X20TB12e : X20TB12 v1.0.0.0
```

### Config.mappmotioncfg - 5PC900_TS17_00/mappMotion/Config.mappmotioncfg
```
Element MappMotionConfiguration (Type=mappmotioncfg)
  Processing:
    ProcessingTaskClass = 1
    ExplicitComputationOrder:
      Axis = NotUsed
  Logger:
    SelectiveLogging = NotUsed
  SharedAlarms:
    Axis = NotUsed
    ACOPOSmultiAuxiliarySupplyModule = NotUsed
    ACOPOSmultiPowerSupplyModule = NotUsed
    AxesGroup = NotUsed
    Assembly = NotUsed
    Segment = NotUsed
    Sector = NotUsed
    Shuttle = NotUsed
    CamOperations = NotUsed
  McAcpDrv:
    POWERLINKCyclesPerParID = 2
```

### Config_1.assembly - 5PC900_TS17_00/mappMotion/Config_1.assembly
```
Element gAssembly_1 (Type=assembly)
  Tracks:
    TrackSeparation = 0.030
    Track[1]:
      Segments:
        SegmentRef[1] = gSegA1
        SegmentRef[2] = gSegA14
        SegmentRef[3] = gSegA13
        SegmentRef[4] = gSegA12
        SegmentRef[5] = gSegA11
        SegmentRef[6] = gSegA10
        SegmentRef[7] = gSegA9
        SegmentRef[8] = gSegA8
        SegmentRef[9] = gSegA7
        SegmentRef[10] = gSegA6
        SegmentRef[11] = gSegA5
        SegmentRef[12] = gSegA4
        SegmentRef[13] = gSegA3
        SegmentRef[14] = gSegA2
      Position = Absolute
        SegmentRef = gSegA1
        SegmentCountDirection = RightToLeft
        Translation:
          X = 0.0
          Y = 0.0
          Z = 0.0
        Orientation:
          Angle1 = 0.0
          Angle2 = 0.0
          Angle3 = 0.0
    Track[2]:
      Segments:
        SegmentRef[1] = ::gSegB5
        SegmentRef[2] = ::gSegB4
        SegmentRef[3] = ::gSegB3
        SegmentRef[4] = ::gSegB2
        SegmentRef[5] = ::gSegB1
        SegmentRef[6] = ::gSegB18
        SegmentRef[7] = ::gSegB17
      Position = RelativeToOne
        TrackSegmentPosition:
          SegmentRef = ::gSegB18
        Base:
          SegmentRef = ::gSegA2
          PositionRelativeTo = FromEnd
    Track[3]:
      Segments:
        SegmentRef[1] = ::gSegB15
        SegmentRef[2] = ::gSegB16
      Position = RelativeToOne
        TrackSegmentPosition:
          SegmentRef = ::gSegB16
          PositionRelativeTo = FromEnd
        Base:
          SegmentRef = ::gSegB17
          Position = 0.09
          PositionRelativeTo = FromEnd
    Track[4]:
      Segments:
        SegmentRef[1] = ::gSegB14
        SegmentRef[2] = ::gSegB13
        SegmentRef[3] = ::gSegB12
        SegmentRef[4] = ::gSegB11
        SegmentRef[5] = ::gSegB10
        SegmentRef[6] = ::gSegB9
        SegmentRef[7] = ::gSegB8
      Position = RelativeToOne
        TrackSegmentPosition:
          SegmentRef = ::gSegB14
        Base:
          SegmentRef = ::gSegB15
          Position = 0.09
    Track[5]:
      Segments:
        SegmentRef[1] = ::gSegB6
        SegmentRef[2] = ::gSegB7
      Position = RelativeToOne
        TrackSegmentPosition:
          SegmentRef = ::gSegB6
        Base:
          SegmentRef = ::gSegB5
          Position = 0.09
  CommonSegmentSettings:
    SegmentSimulationOnPLC = On
    CoggingCompensation = Active
      UpperVelLimit = 0.5
    ElongationCompensation = Inactive
    StopReaction = InductionHalt
    SpeedFilter = NotUsed
    ControllerParameters:
      DefaultParameter:
        Controller:
          Position:
            ProportionalGain = 0.0
          Speed:
            ProportionalGain = 0.0
            IntegrationTime = 0.0
          FeedForward:
            TotalMass = 0.0
            ForcePositive = 0.0
            ForceNegative = 0.0
            SpeedForceFactor = 0.0
            ForceLoad = 0.0
        MovementErrorLimits:
          PositionError = 0.004
          VelocityError = 1.2
        Diverter:
          ForceOverride = 1.0
      AdditionalParameterSets = NotUsed
    ScopeOfErrorReaction = Assembly
    ShuttleIdentificationTime = 0
    PositionControllerLagMonitor = Inactive
    Diverter:
      DiverterWeakEndOverrideFactor = 1.0
      DiverterStrenEndOverrideFactor = 1.0
  Shuttles:
    MaxShuttleCount = 50
    MaxShuttleCommandCount = 0
    Deceleration = 0.0
    UseConvoys = Inactive
    SwitchSectorAfterStop = SwitchOntoSegmentSector
      Scope = ShSs
    DistanceReserve:
      Collision = 0.002
      ErrorStop = 0.006
    ShuttleStereotypes:
      ShuttleStRef[1] = ShuttleStereotype_1
    MagnetPlateConfigurations:
      ShuttleType[1] = 8F1SA.100.xxxxxx-x
    CollisionAvoidance:
      Strategy = Constant
      Exclusion = NotUsed
      MaximumModelDimensions:
        Length:
          ExtentToFront = 0.025
          ExtentToBack = 0.025
        Width:
          Width = 0.046
    Coupling:
      CouplingFeature:
        EliminateShuttleToShuttleDelay = FALSE
  Visualization:
    MonitoringPv
    ProcessingTaskClass = 4
  Alarms = None
Element gAssembly_2 (Type=assembly)
  Tracks:
    TrackSeparation = 0.030
    Track[1]:
      Segments:
        SegmentRef[1] = ::gSegC2
        SegmentRef[2] = ::gSegC3
        SegmentRef[3] = ::gSegC4
        SegmentRef[4] = ::gSegC5
        SegmentRef[5] = ::gSegC6
        SegmentRef[6] = ::gSegC7
        SegmentRef[7] = ::gSegC8
        SegmentRef[8] = ::gSegC9
        SegmentRef[9] = ::gSegC10
        SegmentRef[10] = ::gSegC11
        SegmentRef[11] = ::gSegC12
        SegmentRef[12] = ::gSegC1
      Position = Absolute
        SegmentRef = ::gSegC2
        SegmentCountDirection = RightToLeft
        Translation:
          X = 0.0
          Y = 0.0
          Z = 0.0
        Orientation:
          Angle1 = 0.0
          Angle2 = 0.0
          Angle3 = 0.0
  CommonSegmentSettings:
    SegmentSimulationOnPLC = On
    CoggingCompensation = Active
      UpperVelLimit = 0.5
    ElongationCompensation = Inactive
    StopReaction = InductionHalt
    SpeedFilter = NotUsed
    ControllerParameters:
      DefaultParameter:
        Controller:
          Position:
            ProportionalGain = 0.0
          Speed:
            ProportionalGain = 0.0
            IntegrationTime = 0.0
          FeedForward:
            TotalMass = 0.0
            ForcePositive = 0.0
            ForceNegative = 0.0
            SpeedForceFactor = 0.0
            ForceLoad = 0.0
        MovementErrorLimits:
          PositionError = 0.004
          VelocityError = 1.2
        Diverter:
          ForceOverride = 1.0
      AdditionalParameterSets = NotUsed
    ScopeOfErrorReaction = Assembly
    ShuttleIdentificationTime = 0
    PositionControllerLagMonitor = Inactive
    Diverter:
      DiverterWeakEndOverrideFactor = 1.0
      DiverterStrenEndOverrideFactor = 1.0
  Shuttles:
    MaxShuttleCount = 50
    MaxShuttleCommandCount = 0
    Deceleration = 0.0
    UseConvoys = Inactive
    SwitchSectorAfterStop = SwitchOntoSegmentSector
      Scope = ShSs
    DistanceReserve:
      Collision = 0.002
      ErrorStop = 0.006
    ShuttleStereotypes:
      ShuttleStRef[1] = ShuttleStereotype_1
    MagnetPlateConfigurations:
      ShuttleType[1] = 8F1SA.100.xxxxxx-x
    CollisionAvoidance:
      Strategy = Constant
      Exclusion = NotUsed
      MaximumModelDimensions:
        Length:
          ExtentToFront = 0.025
          ExtentToBack = 0.025
        Width:
          Width = 0.046
    Coupling:
      CouplingFeature:
        EliminateShuttleToShuttleDelay = FALSE
  Visualization:
    MonitoringPv
    ProcessingTaskClass = 4
  Alarms = None
```

### Config_2.shuttlestereotype - 5PC900_TS17_00/mappMotion/Config_2.shuttlestereotype
```
Element ShuttleStereotype_1 (Type=shuttlestereotype)
  MeasurementUnit = 5067858
  MeasurementResolution = 0.00001
  MovementLimits = Internal
    VelocityIsReadOnly = 0
    Velocity:
      Velocity = 4.0
    AccelerationIsReadOnly = 0
    Acceleration:
      Acceleration = 10.0
    DecelerationIsReadOnly = 0
    Deceleration:
      Deceleration = 10.0
    UpdateMode = Immediately
  JerkFilter = Used
    JerkTime = 0.02
  UserData:
    Size = 0
  StateTransitions:
    AutomaticRecontrol = Active
```

### Config_3.sector - 5PC900_TS17_00/mappMotion/Config_3.sector
```
Element gSecOvalA (Type=sector)
  Type = Composed
    StartSegment:
      SegmentRef = ::gSegA1
    IntermediateSegments:
      SegmentRef[1] = ::gSegA14
      SegmentRef[2] = ::gSegA13
      SegmentRef[3] = ::gSegA12
      SegmentRef[4] = ::gSegA11
      SegmentRef[5] = ::gSegA10
      SegmentRef[6] = ::gSegA9
      SegmentRef[7] = ::gSegA8
      SegmentRef[8] = ::gSegA7
      SegmentRef[9] = ::gSegA6
      SegmentRef[10] = ::gSegA5
      SegmentRef[11] = ::gSegA4
      SegmentRef[12] = ::gSegA3
    EndSegment:
      SegmentRef = ::gSegA2
      PositionRelativeTo = FromEnd
  Alarms = None
Element gSecOvalB (Type=sector)
  Type = Composed
    StartSegment:
      SegmentRef = ::gSegB1
      PositionRelativeTo = FromEnd
    IntermediateSegments:
      SegmentRef[1] = ::gSegB2
      SegmentRef[2] = ::gSegB3
      SegmentRef[3] = ::gSegB4
      SegmentRef[4] = ::gSegB5
      SegmentRef[5] = ::gSegB6
      SegmentRef[6] = ::gSegB7
      SegmentRef[7] = ::gSegB8
      SegmentRef[8] = ::gSegB9
      SegmentRef[9] = ::gSegB10
      SegmentRef[10] = ::gSegB11
      SegmentRef[11] = ::gSegB12
      SegmentRef[12] = ::gSegB13
      SegmentRef[13] = ::gSegB14
      SegmentRef[14] = ::gSegB15
      SegmentRef[15] = ::gSegB16
      SegmentRef[16] = ::gSegB17
    EndSegment:
      SegmentRef = ::gSegB18
  Alarms = None
Element gSecCompleteLoop1 (Type=sector)
  Type = Composed
    StartSegment:
      SegmentRef = ::gSegA1
    IntermediateSegments:
      SegmentRef[1] = ::gSegA14
      SegmentRef[2] = ::gSegA13
      SegmentRef[3] = ::gSegA12
      SegmentRef[4] = ::gSegA11
      SegmentRef[5] = ::gSegA10
      SegmentRef[6] = ::gSegA9
      SegmentRef[7] = ::gSegA8
      SegmentRef[8] = ::gSegA7
      SegmentRef[9] = ::gSegA6
      SegmentRef[10] = ::gSegA5
      SegmentRef[11] = ::gSegA4
      SegmentRef[12] = ::gSegA3
      SegmentRef[13] = ::gSegA2
      SegmentRef[14] = ::gSegB1
      SegmentRef[15] = ::gSegB2
      SegmentRef[16] = ::gSegB3
      SegmentRef[17] = ::gSegB4
      SegmentRef[18] = ::gSegB5
      SegmentRef[19] = ::gSegB6
      SegmentRef[20] = ::gSegB7
      SegmentRef[21] = ::gSegB8
      SegmentRef[22] = ::gSegB9
      SegmentRef[23] = ::gSegB10
      SegmentRef[24] = ::gSegB11
      SegmentRef[25] = ::gSegB12
      SegmentRef[26] = ::gSegB13
      SegmentRef[27] = ::gSegB14
      SegmentRef[28] = ::gSegB15
      SegmentRef[29] = ::gSegB16
      SegmentRef[30] = ::gSegB17
    EndSegment:
      SegmentRef = ::gSegB18
  Alarms = None
Element gSecOvalC (Type=sector)
  Type = Composed
    StartSegment:
      SegmentRef = ::gSegC2
    IntermediateSegments:
      SegmentRef[1] = ::gSegC3
      SegmentRef[2] = ::gSegC4
      SegmentRef[3] = ::gSegC5
      SegmentRef[4] = ::gSegC6
      SegmentRef[5] = ::gSegC7
      SegmentRef[6] = ::gSegC8
      SegmentRef[7] = ::gSegC9
      SegmentRef[8] = ::gSegC10
      SegmentRef[9] = ::gSegC11
      SegmentRef[10] = ::gSegC12
    EndSegment:
      SegmentRef = ::gSegC1
      PositionRelativeTo = FromEnd
  Alarms = None
```

### Config_4.processpoint - 5PC900_TS17_00/mappMotion/Config_4.processpoint
```
Element PP_ErrorPosition1 (Type=processpoint)
  Type = AcpTrakPoint
    SectorRef = gSecB7
    Position = 0.2
    TriggerEventBufferSize = 10
    BarrierFunctionality = Off
Element PP_ErrorPosition2 (Type=processpoint)
  Type = AcpTrakPoint
    SectorRef = gSecC7
    Position = 0.1
    TriggerEventBufferSize = 10
    BarrierFunctionality = Off
```

### Config_4.processpointlist - 5PC900_TS17_00/mappMotion/Config_4.processpointlist
```
Element ProcessPointList_1 (Type=processpointlist)
  ProcessPoint[0]:
    Name = PP_ErrorPosition1
    SectorRef = gSecB7
    Position = 0.2
    TriggerEventBufferSize = 10
    BarrierFunctionality = Off
Element ProcessPointList_2 (Type=processpointlist)
  ProcessPoint[0]:
    Name = PP_ErrorPosition2
    SectorRef = gSecC7
    Position = 0.1
    TriggerEventBufferSize = 10
    BarrierFunctionality = Off
```

## Logical view

Binary libraries used (declarations not repeated): operator, runtime, astime, AsIecCon, AsZip, FileIO, standard, AsBrStr, sys_lib, brsystem, ArEventLog, DataObj, AsHttp, AsArSdm, MpBase 6.1.0, McBase 6.0.0, McAcpAx 5.26.1, McAxis 6.0.0, MpAxis 5.26.1, McAcpTrak 6.0.0, CoTrace 6.0.2, TrakDiag

### Package Logical/Libraries - Global libraries

### Segments.var
```iecst
VAR
	gSegA1 : McSegmentType;
	gSegA2 : McSegmentType;
	gSegA3 : McSegmentType;
	gSegA4 : McSegmentType;
	gSegA5 : McSegmentType;
	gSegA6 : McSegmentType;
	gSegA7 : McSegmentType;
	gSegA8 : McSegmentType;
	gSegA9 : McSegmentType;
	gSegA10 : McSegmentType;
	gSegA11 : McSegmentType;
	gSegA12 : McSegmentType;
	gSegA13 : McSegmentType;
	gSegA14 : McSegmentType;
	gSegB1 : McSegmentType;
	gSegB2 : McSegmentType;
	gSegB3 : McSegmentType;
	gSegB4 : McSegmentType;
	gSegB5 : McSegmentType;
	gSegB6 : McSegmentType;
	gSegB7 : McSegmentType;
	gSegB8 : McSegmentType;
	gSegB9 : McSegmentType;
	gSegB10 : McSegmentType;
	gSegB11 : McSegmentType;
	gSegB12 : McSegmentType;
	gSegB13 : McSegmentType;
	gSegB14 : McSegmentType;
	gSegB15 : McSegmentType;
	gSegB16 : McSegmentType;
	gSegB17 : McSegmentType;
	gSegB18 : McSegmentType;
	gSegC1 : McSegmentType;
	gSegC2 : McSegmentType;
	gSegC3 : McSegmentType;
	gSegC4 : McSegmentType;
	gSegC5 : McSegmentType;
	gSegC6 : McSegmentType;
	gSegC7 : McSegmentType;
	gSegC8 : McSegmentType;
	gSegC9 : McSegmentType;
	gSegC10 : McSegmentType;
	gSegC11 : McSegmentType;
	gSegC12 : McSegmentType;
END_VAR
```

### Assembly.typ
```iecst
TYPE
	AssemblyStepEnum :
		(
		ASM_INIT,
		ASM_GET_INFO,
		ASM_W_READY_FOR_POWER_ON,
		ASM_POWER_IS_OFF,
		ASM_W_POWER_ON,
		ASM_ADD_SIM_SHUTTLES,
		ASM_POWER_IS_ON := 100,
		ASM_START_MOVEMENT,
		ASM_W_POWER_OFF,
		ASM_SIMULATE_ERROR,
		ASM_WAIT_FOR_DEFECT_SHUTTLE,
		ASM_ERR_GET_INFO := 9000,
		ASM_ERR_POWERING_ON,
		ASM_ERR_POWERING_OFF,
		ASM_ERR_START_MOVEMENT,
		ASM_ERR_ADDING_SHUTTLE,
		ASM_ERR_SIMULATE_ERROR,
		ASM_ERR_GENERAL
		);
	AssemblyResetStepEnum :
		(
		ASMR_NO_ERROR,
		ASMR_W_ACKNOWLEDGE,
		ASMR_RESET,
		ASMR_INTERNAL_ERROR
		);
	AssemblyStatusType : 	STRUCT
		Step : AssemblyStepEnum;
		ResetStep : AssemblyResetStepEnum;
		AllShuttlesMoving : BOOL;
		Disabled : BOOL;
		Ready : BOOL;
		Homing : BOOL;
		Stopping : BOOL;
		ErrorStop : BOOL;
		SimulationOnPlcMode : McAcpTrakSimulationOnPlcEnum;
		Info : McAcpTrakAsmInfoType;
	END_STRUCT;
	AssemblyParaType : 	STRUCT
		NumberOfSimulatedShuttles : USINT;
	END_STRUCT;
	AssemblyCmdType : 	STRUCT
		Reset : BOOL;
		PowerOn : BOOL;
		PowerOff : BOOL;
		Start : BOOL;
		SimEncoderError : BOOL;
		SimChannelError : BOOL;
		SimSegmentError : BOOL;
	END_STRUCT;
	AssemblyType : 	STRUCT
		SizeOf : UDINT; (*size of this struct*)
		Status : AssemblyStatusType;
		Para : AssemblyParaType;
		Cmd : AssemblyCmdType;
	END_STRUCT;
END_TYPE
```

### Library Logical/Trak/Libraries/TrakLib (IEC, version 0.00.0)
Depends on: standard, AsBrStr

#### Constants.var - Exported constants
```iecst
VAR CONSTANT
	TL_MAX_SHUTTLE : UINT := 199; (* *) (* *) (*#OMIT*)
END_VAR
```

#### Types.typ - Exported data types
```iecst
TYPE
	TL_ShWheelChkData_Type : 	STRUCT
		ShuttleAxis : McAxisType;
		PeakLagError : LREAL; (*maximum lag error*)
		AverageLagError : LREAL; (*average lag error*)
		Good : BOOL; (*shuttle wheels in good condition*)
		Bad : BOOL; (*shuttle wheels in bad condition*)
	END_STRUCT;
END_TYPE
```

#### TrakLib.fun - Exported functions and function blocks
```iecst
{REDUND_ERROR} {REDUND_UNREPLICABLE} FUNCTION_BLOCK TL_StartShuttlesInSector (*starts all shuttles in a given sector*) (*$GROUP=User,$CAT=User,$GROUPICON=User.png,$CATICON=User.png*)
	VAR_INPUT
		Execute : {REDUND_UNREPLICABLE} BOOL;
		Sector : {REDUND_UNREPLICABLE} McSectorType; (*shuttles on this sector should be moved*)
		StartPosition : {REDUND_UNREPLICABLE} LREAL; (*Start of the sector section where the shuttles to be output are located
The starting position must be between 0 and the length of the sector. If not set, value 0 is used.*)
		EndPosition : {REDUND_UNREPLICABLE} LREAL; (*End of the sector section on which the shuttles to be output are located
The end position must be between 0 and the length of the sector. If not set or set to 0, the length of the sector is used.*)
		TargetSector : {REDUND_UNREPLICABLE} McSectorType; (*target sector. If not given then only a velocity command is started*)
		Position : {REDUND_UNREPLICABLE} LREAL; (*position on target sector. Will be ignored if TargetSector is not given*)
		Absolute : {REDUND_UNREPLICABLE} BOOL; (*absolute movement if set*)
		Velocity : {REDUND_UNREPLICABLE} REAL;
		Direction : {REDUND_UNREPLICABLE} McDirectionEnum; (*move all shuttles forward (positive direction)*)
		Acceleration : {REDUND_UNREPLICABLE} REAL;
		Deceleration : {REDUND_UNREPLICABLE} REAL;
		Jerk : {REDUND_UNREPLICABLE} REAL;
	END_VAR
	VAR_OUTPUT
		NumberOfShuttles : {REDUND_UNREPLICABLE} USINT;
		Done : {REDUND_UNREPLICABLE} BOOL;
		Busy : {REDUND_UNREPLICABLE} BOOL;
		Error : {REDUND_UNREPLICABLE} BOOL;
		ErrorID : {REDUND_UNREPLICABLE} UDINT;
	END_VAR
	VAR
		n : {REDUND_UNREPLICABLE} USINT;
		list : {REDUND_UNREPLICABLE} ARRAY[0..255] OF McAxisType; (*the list of shuttles*)
		step : {REDUND_UNREPLICABLE} UINT;
		fbSecGetShuttle : {REDUND_UNREPLICABLE} MC_BR_SecGetShuttle_AcpTrak;
		fbRoutedMoveVel : {REDUND_UNREPLICABLE} MC_BR_RoutedMoveVel_AcpTrak;
		fbRoutedMoveAbs : {REDUND_UNREPLICABLE} MC_BR_RoutedMoveAbs_AcpTrak;
		fbReset : {REDUND_UNREPLICABLE} MC_Reset;
		fbSecReadInfo : {REDUND_UNREPLICABLE} MC_BR_SecReadInfo_AcpTrak;
		ton : {REDUND_UNREPLICABLE} TON;
		maxShuttles : {REDUND_UNREPLICABLE} UINT;
	END_VAR
END_FUNCTION_BLOCK

{REDUND_ERROR} {REDUND_UNREPLICABLE} FUNCTION_BLOCK TL_Barrier (*open/ close a barrier*) (*$GROUP=User,$CAT=User,$GROUPICON=User.png,$CATICON=User.png*)
	VAR_INPUT
		Enable : {REDUND_UNREPLICABLE} BOOL;
		Close : {REDUND_UNREPLICABLE} BOOL;
		ProcessPoint : {REDUND_UNREPLICABLE} McProcessPointType;
	END_VAR
	VAR_OUTPUT
		BarrierClosed : {REDUND_UNREPLICABLE} BOOL;
		BarrierOpen : {REDUND_UNREPLICABLE} BOOL;
		Error : {REDUND_UNREPLICABLE} BOOL;
		ErrorID : {REDUND_UNREPLICABLE} DINT;
	END_VAR
	VAR
		MC_BR_BarrierCommand : {REDUND_UNREPLICABLE} MC_BR_BarrierCommand_AcpTrak;
		MC_BR_BarrierReadInfo : {REDUND_UNREPLICABLE} MC_BR_BarrierReadInfo_AcpTrak;
	END_VAR
END_FUNCTION_BLOCK

{REDUND_ERROR} {REDUND_UNREPLICABLE} FUNCTION_BLOCK TL_CatchShuttle (*catches a shuttle at a process point*) (*$GROUP=User,$CAT=User,$GROUPICON=User.png,$CATICON=User.png*)
	VAR_INPUT
		Enable : {REDUND_UNREPLICABLE} BOOL;
		ProcessPoint : {REDUND_UNREPLICABLE} McProcessPointType; (*process point at entry*)
		DataAddress : {REDUND_UNREPLICABLE} UDINT; (*pointer to variable for shuttle's user data*)
		DataSize : {REDUND_UNREPLICABLE} UDINT; (*sizeof shuttle's user data*)
	END_VAR
	VAR_OUTPUT
		Busy : {REDUND_UNREPLICABLE} BOOL;
		Valid : {REDUND_UNREPLICABLE} BOOL;
		Error : {REDUND_UNREPLICABLE} BOOL;
		ErrorID : {REDUND_UNREPLICABLE} DINT;
		ShuttleCounter : {REDUND_UNREPLICABLE} DINT; (*shuttle counter at exit process point*)
		Axis : {REDUND_UNREPLICABLE} McAxisType;
		ShuttleInfo : {REDUND_UNREPLICABLE} McAcpTrakShInfoType;
	END_VAR
	VAR
		fbTrgPointEnableEntry : {REDUND_UNREPLICABLE} MC_BR_TrgPointEnable_AcpTrak;
		fbTrgPointReadInfo : {REDUND_UNREPLICABLE} MC_BR_TrgPointReadInfo_AcpTrak;
		fbShReadInfo : {REDUND_UNREPLICABLE} MC_BR_ShReadInfo_AcpTrak;
		fbCopyUserData : {REDUND_UNREPLICABLE} MC_BR_ShCopyUserData_AcpTrak;
		step : {REDUND_UNREPLICABLE} UINT;
	END_VAR
END_FUNCTION_BLOCK

{REDUND_ERROR} {REDUND_UNREPLICABLE} FUNCTION_BLOCK TL_ShWheelChk (*Shuttle Wheel Check*) (*$GROUP=User,$CAT=User,$GROUPICON=User.png,$CATICON=User.png*)
	VAR_INPUT
		Enable : {REDUND_UNREPLICABLE} BOOL;
		CycleTime : {REDUND_UNREPLICABLE} LREAL; (*cycle time [s]*)
		CtrlParIndex : {REDUND_UNREPLICABLE} USINT; (*controller settings parameter index for weaking while measurement ( 0 = default )*)
		MeasuringDistance : {REDUND_UNREPLICABLE} LREAL; (*measuring distance (= bumper width) [m]*)
		Threshold : {REDUND_UNREPLICABLE} LREAL; (*lag error threshold for worn shuttle [m]*)
		TrgPointEntry : {REDUND_UNREPLICABLE} McProcessPointType; (*process point at entry*)
		Sector : {REDUND_UNREPLICABLE} McSectorType;
	END_VAR
	VAR_OUTPUT
		Busy : {REDUND_UNREPLICABLE} BOOL;
		Done : {REDUND_UNREPLICABLE} BOOL;
		Error : {REDUND_UNREPLICABLE} BOOL;
		ErrorID : {REDUND_UNREPLICABLE} DINT;
		ShuttleCounter : {REDUND_UNREPLICABLE} DINT; (*shuttle counter at exit process point*)
		Data : {REDUND_UNREPLICABLE} TL_ShWheelChkData_Type;
	END_VAR
	VAR
		fbTrgPointEnableEntry : {REDUND_UNREPLICABLE} MC_BR_TrgPointEnable_AcpTrak;
		fbTrgPointReadInfo : {REDUND_UNREPLICABLE} MC_BR_TrgPointReadInfo_AcpTrak;
		fbShReadInfo : {REDUND_UNREPLICABLE} MC_BR_ShReadInfo_AcpTrak;
		fbShReadSegmentInfo : {REDUND_UNREPLICABLE} MC_BR_ShReadSegmentInfo_AcpTrak;
		fbShReadSectorPos : {REDUND_UNREPLICABLE} MC_BR_ShReadSectorPos_AcpTrak;
		fbShSelCtrlParSet : {REDUND_UNREPLICABLE} MC_BR_ShSelCtrlParSet_AcpTrak;
		currentLagError : {REDUND_UNREPLICABLE} LREAL; (*current lag error with cycle time compensation*)
		setPosDelay : {REDUND_UNREPLICABLE} ARRAY[0..5] OF LREAL; (*fifo for cycle time compensation*)
		n : {REDUND_UNREPLICABLE} UINT;
		l : {REDUND_UNREPLICABLE} LREAL; (*temporary variable*)
		cycleCount : {REDUND_UNREPLICABLE} UDINT; (*cycle counter, starts when a shuttle enters and stops when shuttle leaves*)
		step : {REDUND_UNREPLICABLE} UINT;
		tonTimeout : {REDUND_UNREPLICABLE} TON; (*timeout if shuttle enters but does not leave*)
		start_position : {REDUND_UNREPLICABLE} LREAL; (*sector position where measurement starts*)
		end_position : {REDUND_UNREPLICABLE} LREAL; (*sector position where measurement stops*)
		peakLagError : {REDUND_UNREPLICABLE} LREAL;
		lagErrorSum : {REDUND_UNREPLICABLE} LREAL;
	END_VAR
	VAR CONSTANT
		CYCLES_PLK : UINT := 6; (*total number of cycles for PLK delay*)
	END_VAR
	VAR
		axis : {REDUND_UNREPLICABLE} McAxisType;
		timeouts : {REDUND_UNREPLICABLE} DINT; (*counter for shuttle timeouts (just for debugging)*)
	END_VAR
END_FUNCTION_BLOCK
```

#### TL_Barrier.st
```iecst
(* TODO: Add your comment here *)
FUNCTION_BLOCK TL_Barrier
	IF Enable THEN

		(* Barrier parameters *)
		MC_BR_BarrierCommand.ProcessPoint := ADR(ProcessPoint);
		MC_BR_BarrierReadInfo.ProcessPoint := ADR(ProcessPoint);
		MC_BR_BarrierReadInfo.Enable := TRUE;
		MC_BR_BarrierReadInfo();

		(* Waiting for a command *)
		IF Close AND (MC_BR_BarrierReadInfo.BarrierInfo.Status = mcACPTRAK_BARRIER_OPENED ) THEN
			MC_BR_BarrierCommand.Command := mcACPTRAK_BARRIER_CLOSE;
			MC_BR_BarrierCommand.Execute := TRUE;
		ELSIF NOT Close AND (MC_BR_BarrierReadInfo.BarrierInfo.Status = mcACPTRAK_BARRIER_CLOSED) THEN
			MC_BR_BarrierCommand.Command := mcACPTRAK_BARRIER_OPEN;
			MC_BR_BarrierCommand.Execute := TRUE;
		END_IF

		(* When the tickets are added, reset the execute *)
		IF MC_BR_BarrierCommand.Done THEN
			MC_BR_BarrierCommand.Execute := FALSE;
		END_IF

		(* Call the function block *)
		MC_BR_BarrierCommand();

		IF MC_BR_BarrierReadInfo.BarrierInfo.Status = mcACPTRAK_BARRIER_OPENED THEN
			BarrierClosed := FALSE;
			BarrierOpen := TRUE;
		ELSIF MC_BR_BarrierReadInfo.BarrierInfo.Status = mcACPTRAK_BARRIER_CLOSED THEN
			BarrierClosed := TRUE;
			BarrierOpen := FALSE;
		END_IF;

		Error := MC_BR_BarrierCommand.Error;
		ErrorID := MC_BR_BarrierCommand.ErrorID;
	ELSE
		MC_BR_BarrierCommand( Execute := FALSE );
		MC_BR_BarrierReadInfo( Enable := FALSE );
		Error := FALSE;
		ErrorID := 0;
	END_IF
END_FUNCTION_BLOCK
```

#### TL_StartShuttlesInSector.st
```iecst
(*
	starts all shuttles in a given sector

	first of all we get a list of shuttles in a given sector.
	afterwards we execute a elastic movement on all shuttles (optionally stop at the given position)

*)
FUNCTION_BLOCK TL_StartShuttlesInSector

	IF Execute THEN

		CASE step OF

		(* -------------------------------------------------------------------------------------------
		start
		---------------------------------------------------------------------------------------------*)
		0:
		Busy := TRUE;
		brsmemset(ADR(list), 0, SIZEOF(list));
		maxShuttles := SIZEOF(list)/SIZEOF(list[0]);
		fbSecGetShuttle.Sector := ADR(Sector);
		fbSecGetShuttle.AdvancedParameters.SelectionMode := mcACPTRAK_GET_SH_ALL;
		fbSecGetShuttle.AdvancedParameters.VirtualSelectionMode := mcACPTRAK_GET_SH_VIRT_NONVIRTUAL;
		fbSecGetShuttle.AdvancedParameters.StartPosition := StartPosition;
		fbSecGetShuttle.AdvancedParameters.EndPosition := EndPosition;
		fbSecGetShuttle.Next := FALSE;
		fbSecGetShuttle.Enable := TRUE;

		IF Direction = mcDIR_POSITIVE THEN
			fbSecGetShuttle( Mode := mcACPTRAK_SEARCH_BACKWARD );
			fbRoutedMoveVel.AdvancedParameters.ShuttleOrientation := mcDIR_UNDEFINED;
			fbRoutedMoveVel.AdvancedParameters.StartDirection := mcDIR_UNDEFINED;
			fbRoutedMoveVel.AdvancedParameters.EndDirection := mcDIR_POSITIVE;
			fbRoutedMoveAbs.AdvancedParameters.ShuttleOrientation := mcDIR_UNDEFINED;
			fbRoutedMoveAbs.AdvancedParameters.StartDirection := mcDIR_UNDEFINED;
			fbRoutedMoveAbs.AdvancedParameters.EndDirection := mcDIR_POSITIVE;
		ELSE
			fbSecGetShuttle( Mode := mcACPTRAK_SEARCH_FORWARD );
			fbRoutedMoveVel.AdvancedParameters.ShuttleOrientation := mcDIR_UNDEFINED;
			fbRoutedMoveVel.AdvancedParameters.StartDirection := mcDIR_UNDEFINED;
			fbRoutedMoveVel.AdvancedParameters.EndDirection := mcDIR_NEGATIVE;
			fbRoutedMoveAbs.AdvancedParameters.ShuttleOrientation := mcDIR_UNDEFINED;
			fbRoutedMoveAbs.AdvancedParameters.StartDirection := mcDIR_UNDEFINED;
			fbRoutedMoveAbs.AdvancedParameters.EndDirection := mcDIR_NEGATIVE;
		END_IF

		IF fbSecGetShuttle.Valid THEN
			NumberOfShuttles := UINT_TO_USINT(fbSecGetShuttle.TotalCount);
			IF NumberOfShuttles > 0 THEN

				list[0] := fbSecGetShuttle.Axis;

				IF fbSecGetShuttle.RemainingCount > 0 THEN (* more then one shuttle *)
					n := 1;
					fbSecGetShuttle( Next := TRUE );
					step := 10;
				ELSE (* only one shuttle *)
					fbSecGetShuttle( Enable	:= FALSE );
					n := 0;
					step := 20;
				END_IF
			ELSE (* no shuttles to start *)
				fbSecGetShuttle( Enable	:= FALSE );
				step := 100;
			END_IF
		ELSIF fbSecGetShuttle.Error THEN
			Error := TRUE;
			ErrorID := step;
			step := 9001; (* error *)
		ELSE
			fbSecGetShuttle();
		END_IF;

		(* -------------------------------------------------------------------------------------------
		get the list of shuttles in sector
		---------------------------------------------------------------------------------------------*)
		10:
		IF 	fbSecGetShuttle.Axis.controlif <> list[n-1].controlif THEN
			IF fbSecGetShuttle.Error THEN
				Error := TRUE;
				ErrorID := step;
				fbSecGetShuttle( Enable := FALSE );
				step := 9002; (* error *)
			ELSE
				fbSecGetShuttle( Next := FALSE );
				list[n] := fbSecGetShuttle.Axis;
				n := n + 1;
				IF (fbSecGetShuttle.RemainingCount > 0) AND (n < maxShuttles) THEN
						fbSecGetShuttle( Next := TRUE );
				ELSE (* all shuttles found *)
					n := 0;
					fbSecGetShuttle( Enable := FALSE );
					step := 20;
				END_IF
			END_IF
		ELSE
			fbSecGetShuttle();
		END_IF

		(* -------------------------------------------------------------------------------------------
		reset shuttle
		---------------------------------------------------------------------------------------------*)
	    20:
		fbReset( Axis := ADR(list[n]), Execute := TRUE );
		IF fbReset.Done THEN
			fbReset( Execute := FALSE );
			n := n + 1;
			IF n < maxShuttles THEN
				IF list[n].controlif = 0 THEN (* all shuttles reset *)
					fbSecReadInfo( Sector := ADR(Sector), Enable := FALSE ); (* reset fb *)
					ton( PT := T#1s, IN := FALSE ); (* reset fb *)
					step := 30;
				END_IF
			ELSE (* end of list *)
				fbSecReadInfo( Sector := ADR(Sector), Enable := FALSE ); (* reset fb *)
				ton( PT := T#1s, IN := FALSE ); (* reset fb *)
				step := 30;
			END_IF
		ELSIF fbReset.Error THEN
			Error := TRUE;
			ErrorID := step;
			step := 9003; (* error *)
		ELSE
			fbReset();
		END_IF

		(* -------------------------------------------------------------------------------------------
		wait until no shuttle is in 'Disabled' state (or timeout has expired )
		---------------------------------------------------------------------------------------------*)
		30:
		fbSecReadInfo( Enable := TRUE );
		ton( IN := TRUE );
		IF ton.Q THEN
			fbSecReadInfo( Sector := ADR(Sector), Enable := FALSE ); (* reset fb *)
			ton( PT := T#1s, IN := FALSE ); (* reset fb *)
			n := 0;
			step := 40;
		ELSIF fbSecReadInfo.Valid THEN
			IF fbSecReadInfo.SectorInfo.ShuttleCount.InDisabled = 0 THEN
				fbSecReadInfo( Sector := ADR(Sector), Enable := FALSE ); (* reset fb *)
				ton( PT := T#1s, IN := FALSE ); (* reset fb *)
				n := 0;
				step := 40;
			END_IF
		ELSIF fbSecReadInfo.Error THEN
			fbSecReadInfo( Enable := FALSE ); (* reset fb *)
			Error := TRUE;
			ErrorID := step;
			step := 9006;
		END_IF

		(* -------------------------------------------------------------------------------------------
		start Shuttle
		---------------------------------------------------------------------------------------------*)
		40:
		IF Absolute THEN
			fbRoutedMoveAbs( Axis:= ADR(list[n]), Sector := ADR(TargetSector), Position := Position,
							Velocity := Velocity, Acceleration := Acceleration,
							Deceleration := Deceleration, Jerk := Jerk, BufferMode := mcABORTING, Execute := TRUE );
			step := 70;
		ELSE
			fbRoutedMoveVel( Axis:= ADR(list[n]), Sector := ADR(TargetSector), Position := Position,
							Velocity := Velocity, RouteVelocity := Velocity, Acceleration := Acceleration,
							Deceleration := Deceleration, Jerk := Jerk, BufferMode := mcABORTING, Execute := TRUE );
			step := 50;
		END_IF

		(* -------------------------------------------------------------------------------------------
		wait until movement is started
		---------------------------------------------------------------------------------------------*)
		50:
		IF fbRoutedMoveVel.Active THEN
			fbRoutedMoveVel( Execute := FALSE );
			n := n + 1;
			step := 100; (* assume end of list *)
			IF n < maxShuttles THEN
				IF list[n].controlif <> 0 THEN
					step := 40; (* no, we still need to start a shuttle *)
				END_IF
			END_IF

		ELSIF fbRoutedMoveVel.Error OR fbRoutedMoveVel.CommandAborted THEN
			Error := TRUE;
			ErrorID := step;
			step := 9004; (* error *)
		ELSE
			fbRoutedMoveVel();
		END_IF;

		(* -------------------------------------------------------------------------------------------
		wait until (absolute) movement is started
		---------------------------------------------------------------------------------------------*)
		70:
		IF fbRoutedMoveAbs.Active THEN
			fbRoutedMoveAbs( Execute := FALSE );
			n := n + 1;
			step := 100; (* assume end of list *)
			IF n < maxShuttles THEN
				IF list[n].controlif <> 0 THEN
					step := 40; (* no, we still need to start a shuttle *)
				END_IF
			END_IF
		ELSIF fbRoutedMoveAbs.Error OR fbRoutedMoveAbs.CommandAborted THEN
			Error := TRUE;
			ErrorID := step;
			step := 9005; (* error *)
		ELSE
			fbRoutedMoveAbs();
		END_IF;

		(* -------------------------------------------------------------------------------------------
		done
		---------------------------------------------------------------------------------------------*)
		100:
		Done := TRUE;
		Busy := FALSE;
		Error := FALSE;
		ErrorID := 0;

		(* -------------------------------------------------------------------------------------------
		error
		---------------------------------------------------------------------------------------------*)
		9000..9006: (* Error *)

		END_CASE;

	ELSE
		(* Reset all data if the FUB is disabled *)
		fbSecGetShuttle( Enable	:= FALSE );
		fbRoutedMoveVel( Execute := FALSE );
		fbRoutedMoveAbs( Execute := FALSE );
		fbReset( Execute := FALSE );
		Done					:= FALSE;
		Busy					:= FALSE;
		Error					:= FALSE;
		ErrorID					:= 0;
		NumberOfShuttles		:= 0;
		step		:= 0;
	END_IF

END_FUNCTION_BLOCK
```

#### TL_ShWheelChk.st - Checks the shuttle cover for contact with a segment
```iecst
(* Shuttle Wheel Check *)
FUNCTION_BLOCK TL_ShWheelChk

	IF NOT(Enable) THEN
		step := 0;
	END_IF

	CASE step OF
		(* ------------------------------------------------------------------------------
			wait for Enable
		   ------------------------------------------------------------------------------ *)

		0:
		IF Enable THEN (* activate process points as trigger points *)
			fbTrgPointEnableEntry( ProcessPoint := ADR(TrgPointEntry), Enable := TRUE );
			IF CycleTime < 1200e-6 THEN
				CycleTime := 1200e-6;
			END_IF
			IF fbTrgPointEnableEntry.Valid THEN
				fbTrgPointReadInfo( Execute := FALSE );
				fbShSelCtrlParSet( Execute := FALSE );
				Data.AverageLagError := 0.0;
				Data.PeakLagError := 0.0;
				step := 100;
			ELSIF fbTrgPointEnableEntry.Error THEN
				ErrorID := 1;
				Error := TRUE;
				step := 9000;
			END_IF
		ELSE
			fbShReadInfo( Enable := FALSE );
			fbShReadSectorPos( Enable := FALSE );
			fbShSelCtrlParSet( Execute := FALSE );
			fbTrgPointEnableEntry( Enable := FALSE );
			fbTrgPointReadInfo( Execute := FALSE );
			Done := FALSE;
			Busy := FALSE;
			Error := FALSE;
			ErrorID := 0;
		END_IF

		(* ------------------------------------------------------------------------------
			wait for arriving shuttle at entry trigger point
		   ------------------------------------------------------------------------------ *)

		100:
		fbTrgPointEnableEntry();
		IF fbTrgPointEnableEntry.EventCount <> 0 THEN
			fbTrgPointReadInfo( ProcessPoint := fbTrgPointEnableEntry.ProcessPoint, Execute := TRUE );
			tonTimeout( IN:= FALSE, PT := T#20s ); (* abort timer *)
			tonTimeout.IN := TRUE; (* start timeout *)
			peakLagError := 0.0;
			lagErrorSum := 0.0;
			currentLagError := 0.0;
			Done := FALSE;
			Busy := FALSE;
			step := 110;
		ELSIF fbTrgPointEnableEntry.Error THEN
			ErrorID := 101;
			Error := TRUE;
			step := 9000;
		END_IF

		(* ------------------------------------------------------------------------------
			shuttle passed trigger point - switch on reading shuttle info and reduce
			the controller settings to make the lag error more visible
		   ------------------------------------------------------------------------------ *)

		110:
		IF fbTrgPointReadInfo.Done THEN
			axis := fbTrgPointReadInfo.TrgPointInfo.Axis;
			IF fbTrgPointReadInfo.TrgPointInfo.Event = mcACPTRAK_TP_PASSED_POSITIVE THEN (* only consider shuttles in positive direction *)
				(* switch on reading shuttle info (position) *)
				fbShReadInfo( Axis := ADR(axis), Enable := TRUE );
				(* switch on reading position of sector where triggerpoint is located *)
				fbShReadSectorPos( Axis := ADR(axis), Sector := ADR(Sector), Enable := TRUE );
				(* switch on reading segment info where shuttle is located *)
				fbShReadSegmentInfo( Axis := ADR(axis), Enable := TRUE );
				(* weak position controller to make the lag error more visible *)
				fbShSelCtrlParSet( Axis := ADR(axis), Mode := mcACPTRAK_SIDE_BOTH, ParameterSetIndex := CtrlParIndex, Execute := TRUE );
				step := 120;
			ELSE
				step := 100;
			END_IF
			fbTrgPointReadInfo( Execute := FALSE );
		ELSIF fbTrgPointReadInfo.Busy THEN
			fbTrgPointReadInfo();
		ELSIF fbTrgPointReadInfo.Error THEN
			ErrorID := 111;
			Error := TRUE;
			step := 9000;
		END_IF

		(* ------------------------------------------------------------------------------
			read shuttles's position and lag error (set position - actual position )
		   ------------------------------------------------------------------------------ *)

		120:
		IF fbShReadInfo.Valid AND fbShReadSectorPos.Valid AND fbShReadSegmentInfo.Valid  AND fbShSelCtrlParSet.Done THEN
			cycleCount := 0;
			start_position := fbShReadSectorPos.Info.Position;
			end_position := start_position + MeasuringDistance;
			fbShSelCtrlParSet( Execute := FALSE );
			step := 130;
		ELSIF fbShReadInfo.Error THEN
			ErrorID := 121;
			Error := TRUE;
			step := 9000;
		ELSIF fbShReadSectorPos.Error THEN
			ErrorID := 122;
			Error := TRUE;
			step := 9000;
		ELSIF fbShReadSegmentInfo.Error THEN
			ErrorID := 123;
			Error := TRUE;
			step := 9000;
		ELSIF fbShSelCtrlParSet.Error THEN
			ErrorID := 124;
			Error := TRUE;
			step := 9000;
		ELSE
			fbShReadInfo();
			fbShReadSectorPos();
			fbShSelCtrlParSet();
			fbShReadSegmentInfo();
		END_IF

		(* ------------------------------------------------------------------------------
			read shuttles's position and lag error (set position - actual position )
		   ------------------------------------------------------------------------------ *)

		130:
		(* calculate lag error when fifo is already filled and bumper position is reached *)
		IF  (cycleCount >= CYCLES_PLK) AND (fbShReadSectorPos.Info.Position >= start_position) THEN
			Busy := TRUE;
			l := setPosDelay[0] - fbShReadInfo.ShuttleInfo.CurrentValues.ActualPosition;
			IF l < 0.0001 THEN (* < epsilon or negative *)
				currentLagError := 0.0;
			ELSIF l > 0.008 THEN (* plausibility control at sector end *)
				currentLagError := currentLagError;
			ELSE
				currentLagError := l;
			END_IF
			lagErrorSum := lagErrorSum + currentLagError;
			peakLagError := MAX( peakLagError, currentLagError );
		END_IF
		FOR n := 0 TO (CYCLES_PLK-2) DO (* shift fifo *)
			setPosDelay[n] := setPosDelay[n+1];
		END_FOR
		setPosDelay[CYCLES_PLK-1] := fbShReadInfo.ShuttleInfo.CurrentValues.Position;  (* set position that must be delayed *)

		fbShReadInfo();
		fbShReadSectorPos();
		fbShReadSegmentInfo();

		(* check the exit point to see if the shuttle passed it. *)
		IF (fbShReadSectorPos.Info.Position >= end_position) OR tonTimeout.Q THEN (* shuttle passes exit point *)
			Busy := FALSE;
			(* switch off reading the shuttle position *)
			fbShReadInfo( Enable := FALSE );
			fbShReadSectorPos( Enable := FALSE );
			fbShReadSegmentInfo( Enable := FALSE );
			(* set controller to default again ! *)
			fbShSelCtrlParSet( Axis := ADR(axis), Mode := mcACPTRAK_SIDE_BOTH, ParameterSetIndex := 0, Execute := TRUE );
			IF NOT(tonTimeout.Q) THEN
				Done := TRUE;
				ShuttleCounter := ShuttleCounter + 1; (* a shuttle was measured *)
				Data.ShuttleAxis := axis;
				Data.PeakLagError := peakLagError;
				IF Data.PeakLagError >= ABS(Threshold) THEN
					Data.Good := FALSE;
					Data.Bad := TRUE;
				ELSE
					Data.Good := TRUE;
					Data.Bad := FALSE;
				END_IF
				IF cycleCount <> 0 THEN (* prevent division by zero error *)
					Data.AverageLagError := lagErrorSum / UDINT_TO_LREAL(cycleCount);
				END_IF
			ELSE (* timeout *)
				timeouts := timeouts + 1;  (* just a counter for debugging *)
			END_IF
			step := 140;
		END_IF
		(* count cycles *)
		cycleCount := cycleCount + 1;
		tonTimeout();

		(* ------------------------------------------------------------------------------
			wait until controller settings are on defaults again
		   ------------------------------------------------------------------------------ *)

		140:
		IF 	fbShSelCtrlParSet.Done THEN
			fbShSelCtrlParSet.Execute := FALSE;
			step := 100;
		END_IF
		fbShSelCtrlParSet();

		9000: (* Error *)

	END_CASE

END_FUNCTION_BLOCK
```

#### TL_CatchShuttle.st
```iecst
FUNCTION_BLOCK TL_CatchShuttle

	IF NOT(Enable) THEN
		step := 0;
	END_IF

	CASE step OF
		(* ------------------------------------------------------------------------------
			wait for Enable
		   ------------------------------------------------------------------------------ *)

		0:
		IF Enable THEN (* activate process points as trigger points *)
			Busy := TRUE;
			fbTrgPointEnableEntry.ProcessPoint := ADR(ProcessPoint);
			fbTrgPointEnableEntry.Enable := TRUE;
			step := 100;
		ELSE
			fbShReadInfo( Enable := FALSE );
			fbTrgPointEnableEntry( Enable := FALSE );
			fbTrgPointReadInfo( Execute := FALSE );
			Valid := FALSE;
			Busy := FALSE;
			Error := FALSE;
			ErrorID := 0;
		END_IF

		(* ------------------------------------------------------------------------------
			wait for arriving shuttle at entry trigger point
		   ------------------------------------------------------------------------------ *)

		100:
		fbTrgPointEnableEntry();
		IF fbTrgPointEnableEntry.Valid THEN
			Valid := TRUE;
			IF fbTrgPointEnableEntry.EventCount <> 0 THEN
				fbTrgPointReadInfo( ProcessPoint := fbTrgPointEnableEntry.ProcessPoint, Execute := TRUE );
				step := 110;
			END_IF
		ELSIF fbTrgPointEnableEntry.Error THEN
			Valid := FALSE;
			ErrorID := 101;
			Error := TRUE;
			step := 9000;
		END_IF

		(* ------------------------------------------------------------------------------
			shuttle passed trigger point - switch on reading shuttle info
		   ------------------------------------------------------------------------------ *)

		110:
		IF fbTrgPointReadInfo.Done THEN
			Axis := fbTrgPointReadInfo.TrgPointInfo.Axis;
			IF fbTrgPointReadInfo.TrgPointInfo.Event = mcACPTRAK_TP_PASSED_POSITIVE THEN (* only consider shuttles in positive direction *)
				(* switch on reading shuttle info *)
				fbShReadInfo( Axis := ADR(Axis), Enable := TRUE );
				step := 120;
			ELSE
				step := 100;
			END_IF
			fbTrgPointReadInfo( Execute := FALSE );

		ELSIF fbTrgPointReadInfo.Error THEN
			Valid := FALSE;
			ErrorID := 111;
			Error := TRUE;
			step := 9000;
		ELSE
			fbTrgPointReadInfo();
		END_IF

		(* ------------------------------------------------------------------------------
			read shuttles's info
		   ------------------------------------------------------------------------------ *)

		120:
		IF fbShReadInfo.Valid THEN
			ShuttleInfo := fbShReadInfo.ShuttleInfo;
			fbShReadInfo( Enable := FALSE );
			(* switch on reading shuttle's user data *)
			IF DataAddress <> 0 AND DataSize <> 0 THEN (* shall user data be read, too ? *)
				fbCopyUserData( Axis := ADR(Axis), Mode := mcACPTRAK_USERDATA_GET, DataAddress := DataAddress, DataSize := DataSize, Execute := TRUE );
				step := 130;
			ELSE (* we don't need the user data, so we are ready *)
				ShuttleCounter := ShuttleCounter + 1; (* shuttle data valid *)
				step := 100;
			END_IF
		ELSIF fbShReadInfo.Error THEN
			IF fbShReadInfo.ErrorID = -1067319295 THEN (* ignore 'invalid axis' *)
				fbShReadInfo( Enable := FALSE );
				step := 100;
			ELSE
				Valid := FALSE;
				ErrorID := 121;
				Error := TRUE;
				fbShReadInfo( Enable := FALSE );
				step := 9000;
			END_IF
		ELSE
			fbShReadInfo();
		END_IF

		(* ------------------------------------------------------------------------------
			read shuttles's user data
		   ------------------------------------------------------------------------------ *)

		130:
		IF fbCopyUserData.Done THEN
			fbCopyUserData( Execute := FALSE );
			ShuttleCounter := ShuttleCounter + 1; (* shuttle data valid *)
			step := 100;
		ELSIF fbCopyUserData.Error THEN
			IF fbCopyUserData.ErrorID = -1067319295 THEN (* ignore 'invalid axis' *)
				fbCopyUserData( Execute := FALSE );
				step := 100;
			ELSE
				Valid := FALSE;
				ErrorID := 131;
				Error := TRUE;
				fbCopyUserData( Execute := FALSE );
				step := 9000;
			END_IF
		ELSE
			fbCopyUserData();
		END_IF

		9000: (* Error *)
		Busy := FALSE;

	END_CASE

END_FUNCTION_BLOCK
```

### TrakConstants.var
```iecst
VAR CONSTANT
	TRAK_BASIC_ERROR_ID : DINT := -536870912;
	TRAK_BASIC_SUCCESS_ID : DINT := 536870912;
	TRAK_BASIC_WARNING_ID : DINT := -1610612736;
	TRAK_BASIC_INFO_ID : DINT := 1610612736;
END_VAR
```

### Program Logical/Trak/TrakInit (IEC)

#### Variables.var
```iecst
VAR
	fbLogWrite : TD_LogWrite;
END_VAR
```

#### Main.st
```iecst
PROGRAM _INIT
	(* create the loggers *)
	REPEAT
		fbLogWrite( Name := 'MyTrak', EventID := TRAK_BASIC_SUCCESS_ID, ObjectID := 'MyTrak', Ascii := 'startup', Execute := TRUE );
		UNTIL fbLogWrite.Done OR fbLogWrite.Error
	END_REPEAT
	fbLogWrite( Execute := FALSE );

END_PROGRAM

PROGRAM _CYCLIC
	(* Insert code here *)

END_PROGRAM

PROGRAM _EXIT
	(* Insert code here *)

END_PROGRAM
```

### Program Logical/Trak/AssCtrl1 (IEC)

#### Cyclic.st - Cyclic code
```iecst
PROGRAM _CYCLIC
	(* catch shuttle on gSegB7 for simulation of shuttle errors *)
	fbCatchShuttle();

	(* assembly's state machine *)
	fbLogStep.EventID := TRAK_BASIC_INFO_ID;

	CASE step OF
		ASM_INIT:
		fbGetInfo( Execute := FALSE ); (* reset fb *)
		fbGetInfo( Execute := TRUE );
		fbPowerOn( Execute := FALSE ); (* reset fb *)
		fbPowerOff( Execute := FALSE ); (* reset fb *)
		step := ASM_GET_INFO;

		ASM_GET_INFO:
		fbLogStep.Signal := 'ASM_GET_INFO';
		IF fbGetInfo.Done THEN
			fbGetInfo( Execute := FALSE ); (* reset fb *)
			assemblyCtrl.Status.SimulationOnPlcMode := fbGetInfo.AssemblyInfo.SimulationOnPlcMode;
			step := ASM_W_READY_FOR_POWER_ON;
		ELSIF fbGetInfo.Error THEN
			fbGetInfo( Execute := FALSE ); (* reset fb *)
			step := ASM_ERR_GET_INFO;
			fbLogStep.EventID := TRAK_BASIC_ERROR_ID;
			fbLogStep.Signal := 'ASM_ERR_GET_INFO';
		ELSE (* busy *)
			fbGetInfo();
		END_IF

		ASM_W_READY_FOR_POWER_ON:
		fbLogStep.Signal := 'ASM_W_READY_FOR_POWER_ON';
		IF assemblyCtrl.Status.Info.ReadyForPowerOn THEN
			IF assemblyCtrl.Status.Info.PowerOn THEN
				step := ASM_POWER_IS_ON;
			ELSE
				step := ASM_POWER_IS_OFF;
			END_IF
		END_IF

		ASM_POWER_IS_OFF:
		fbLogStep.Signal := 'ASM_POWER_IS_OFF';
		IF assemblyCtrl.Cmd.PowerOn THEN
			assemblyCtrl.Cmd.PowerOn := FALSE;
			fbPowerOn( Execute := TRUE );
			step := ASM_W_POWER_ON;
		END_IF

		ASM_ADD_SIM_SHUTTLES:
		fbLogStep.Signal := 'ASM_ADD_SIM_SHUTTLES';
		IF fbAddSimShuttle.Done THEN
			fbAddSimShuttle( Execute := FALSE ); (* reset fb *)
			IF assemblyCtrl.Status.Info.ShuttlesCount >= assemblyCtrl.Para.NumberOfSimulatedShuttles OR assemblyCtrl.Para.NumberOfSimulatedShuttles = 0 THEN
				step := ASM_POWER_IS_ON;
			ELSE
				fbAddSimShuttle.Position := fbAddSimShuttle.Position + 0.06;
				fbAddSimShuttle( Execute := TRUE );
			END_IF
		ELSIF fbAddSimShuttle.Error THEN
			fbAddSimShuttle( Execute := FALSE ); (* reset fb *)
			step := ASM_ERR_ADDING_SHUTTLE;
			fbLogStep.EventID := TRAK_BASIC_ERROR_ID;
			fbLogStep.Signal := 'ASM_ERR_ADDING_SHUTTLE';
		ELSE (* busy *)
			fbAddSimShuttle();
		END_IF

		ASM_W_POWER_ON:
		fbLogStep.Signal := 'ASM_W_POWER_ON';
		IF fbPowerOn.Done AND assemblyCtrl.Status.Info.PowerOn THEN
			fbPowerOn( Execute := FALSE );  (* reset fb *)
			IF assemblyCtrl.Status.Info.ShuttlesCount >= assemblyCtrl.Para.NumberOfSimulatedShuttles THEN
				step := ASM_POWER_IS_ON;
			ELSE
				fbAddSimShuttle( Execute := FALSE ); (* reset fb *)
				fbAddSimShuttle( Execute := TRUE );
				step := ASM_ADD_SIM_SHUTTLES;
			END_IF
		ELSIF fbPowerOn.Error THEN
			fbPowerOn( Execute := FALSE );  (* reset fb *)
			step := ASM_ERR_POWERING_ON;
			fbLogStep.EventID := TRAK_BASIC_ERROR_ID;
			fbLogStep.Signal := 'ASM_ERR_POWERING_ON';
		ELSE (* busy *)
			fbPowerOn();
		END_IF

		ASM_POWER_IS_ON:
		fbLogStep.Signal := 'ASM_POWER_IS_ON';
		IF NOT assemblyCtrl.Status.Info.PowerOn THEN
			step := ASM_POWER_IS_OFF;
		ELSIF assemblyCtrl.Cmd.PowerOff THEN
			assemblyCtrl.Cmd.PowerOff := FALSE;
			fbPowerOff( Execute := TRUE );
			step := ASM_W_POWER_OFF;
		ELSIF assemblyCtrl.Cmd.Start THEN
			assemblyCtrl.Cmd.Start := FALSE;
			fbStartShuttles( Execute := FALSE ); (* reset fb *)
			fbStartShuttles( Execute := TRUE ); (* reset fb *)
			step := ASM_START_MOVEMENT;
		ELSIF assemblyCtrl.Cmd.SimSegmentError THEN
			assemblyCtrl.Cmd.SimSegmentError := FALSE;
			fbSegCommandError( Segment := pDefectSegment, Type := TD_SEGERRCMD_SEGMENT, Execute := FALSE ); (* reset fb *)
			fbSegCommandError( Execute := TRUE );
			step := ASM_SIMULATE_ERROR;
		ELSIF assemblyCtrl.Cmd.SimChannelError THEN
			IF assemblyCtrl.Status.AllShuttlesMoving THEN
				assemblyCtrl.Cmd.SimChannelError := FALSE;
				fbSegCommandError( Segment := pDefectSegment, Type := TD_SEGERRCMD_CHANNEL, Execute := FALSE ); (* reset fb *)
				shuttleCounter := fbCatchShuttle.ShuttleCounter;
				step := ASM_WAIT_FOR_DEFECT_SHUTTLE;
			ELSE
				assemblyCtrl.Cmd.SimChannelError := FALSE;
			END_IF
		ELSIF assemblyCtrl.Cmd.SimEncoderError  THEN
			IF assemblyCtrl.Status.AllShuttlesMoving THEN
				assemblyCtrl.Cmd.SimEncoderError := FALSE;
				fbSegCommandError( Segment := pDefectSegment, Type := TD_SEGERRCMD_ENCODER, Execute := FALSE ); (* reset fb *)
				shuttleCounter := fbCatchShuttle.ShuttleCounter;
				step := ASM_WAIT_FOR_DEFECT_SHUTTLE;
			ELSE
				assemblyCtrl.Cmd.SimEncoderError := FALSE;
			END_IF
		END_IF

		ASM_START_MOVEMENT:
		fbLogStep.Signal := 'ASM_START_MOVEMENT';
		IF fbStartShuttles.Done THEN
			fbStartShuttles( Execute := FALSE ); (* reset fb *)
			step := ASM_POWER_IS_ON;
		ELSIF fbStartShuttles.Error THEN
			fbStartShuttles( Execute := FALSE ); (* reset fb *)
			step := ASM_ERR_START_MOVEMENT;
			fbLogStep.EventID := TRAK_BASIC_ERROR_ID;
			fbLogStep.Signal := 'ASM_ERR_START_MOVEMENT';
		ELSE (* busy *)
			fbStartShuttles();
		END_IF

		ASM_SIMULATE_ERROR:
		fbLogStep.Signal := 'ASM_SIMULATE_ERROR';
		IF fbSegCommandError.Done THEN
			fbSegCommandError( Execute := FALSE );
			step := ASM_POWER_IS_ON;
		ELSIF fbSegCommandError.Error THEN
			fbSegCommandError( Execute := FALSE );
			step := ASM_POWER_IS_ON;
//			step := ASM_ERR_SIMULATE_ERROR;
//			fbLogStep.EventID := TRAK_BASIC_ERROR_ID;
//			fbLogStep.Signal := 'ASM_ERR_SIMULATE_ERROR';
		ELSE (* busy *)
			fbSegCommandError();
		END_IF

		ASM_WAIT_FOR_DEFECT_SHUTTLE: (* wait for defect shuttle passing *)
		fbLogStep.Signal := 'ASM_WAIT_FOR_DEFECT_SHUTTLE';
		IF shuttleCounter <> fbCatchShuttle.ShuttleCounter THEN
			fbSegCommandError( Execute := TRUE );
			assemblyCtrl.Cmd.SimChannelError := FALSE;
			assemblyCtrl.Cmd.SimEncoderError := FALSE;
			step := ASM_SIMULATE_ERROR;
		END_IF

		ASM_W_POWER_OFF:
		fbLogStep.Signal := 'ASM_W_POWER_OFF';
		IF fbPowerOff.Done OR  NOT assemblyCtrl.Status.Info.PowerOn THEN
			step := ASM_POWER_IS_OFF;
			fbPowerOff( Execute := FALSE ); (* reset fb *)
		ELSIF fbPowerOff.Error THEN
			fbPowerOff( Execute := FALSE ); (* reset fb *)
			step := ASM_ERR_POWERING_OFF;
			fbLogStep.EventID := TRAK_BASIC_ERROR_ID;
			fbLogStep.Signal := 'ASM_ERR_POWERING_OFF';
		ELSE (* busy *)
			fbPowerOff();
		END_IF

		ASM_ERR_GET_INFO..ASM_ERR_GENERAL:

	END_CASE

	assemblyCtrl.Status.Step := step;
	fbLogStep(); (* log state machine *)

	(* read assembly status *)
	fbReadStatus();
	assemblyCtrl.Status.Disabled  	:= fbReadStatus.AssemblyDisabled;
	assemblyCtrl.Status.ErrorStop 	:= fbReadStatus.AssemblyErrorStop;
	assemblyCtrl.Status.Homing 		:= fbReadStatus.AssemblyHoming;
	assemblyCtrl.Status.Stopping 	:= fbReadStatus.AssemblyStopping;
	assemblyCtrl.Status.Ready 	  	:= fbReadStatus.AssemblyReady;

	(* read assembly info *)
	fbReadInfo();
	assemblyCtrl.Status.Info := fbReadInfo.AssemblyInfo;
	assemblyCtrl.Status.AllShuttlesMoving := FALSE;
	IF assemblyCtrl.Status.Info.ShuttlesCount = assemblyCtrl.Para.NumberOfSimulatedShuttles THEN
		IF assemblyCtrl.Status.Info.ShuttlesInDisabledCount = 0 AND
			assemblyCtrl.Status.Info.ShuttlesInErrorStopCount = 0 AND
			assemblyCtrl.Status.Info.ShuttlesInStandstillCount = 0 AND
			assemblyCtrl.Status.Info.ShuttlesInStoppingCount = 0 THEN
			assemblyCtrl.Status.AllShuttlesMoving := TRUE;
		END_IF
	END_IF

	(* run recorder for breakdown analysis *)
	fbRecorder(Trigger := assemblyCtrl.Status.ErrorStop );
	(* web page *)
	fbWebServices();

	(* reset error stop *)
	fbLogResetStep.EventID := TRAK_BASIC_INFO_ID;
	CASE assemblyCtrl.Status.ResetStep OF
		ASMR_NO_ERROR:
		fbLogResetStep.Signal := 'ASMR_NO_ERROR';
		IF assemblyCtrl.Status.ErrorStop THEN
			fbAsmReset( Execute := FALSE ); (* reset fb *)
			assemblyCtrl.Cmd.Reset := FALSE;
			assemblyCtrl.Status.ResetStep := ASMR_W_ACKNOWLEDGE;
		END_IF

		ASMR_W_ACKNOWLEDGE:
		fbLogResetStep.Signal := 'ASMR_W_ACKNOWLEDGE';
		IF assemblyCtrl.Cmd.Reset THEN
			assemblyCtrl.Cmd.Reset := FALSE;
			fbAsmReset( Execute := TRUE ); (* reset fb *)
			assemblyCtrl.Status.ResetStep := ASMR_RESET;
		END_IF

		ASMR_RESET:
		fbLogResetStep.Signal := 'ASMR_RESET';
		IF fbAsmReset.Done THEN
			fbAsmReset( Execute := FALSE ); (* reset fb *)
			assemblyCtrl.Status.ResetStep := ASMR_NO_ERROR;
		ELSIF fbAsmReset.Error THEN
			fbAsmReset( Execute := FALSE ); (* reset fb *)
			assemblyCtrl.Status.ResetStep := ASMR_INTERNAL_ERROR;
			fbLogResetStep.EventID := TRAK_BASIC_ERROR_ID;
			fbLogResetStep.Signal := 'ASMR_INERNAL_ERROR';
		ELSE (* busy *)
			fbAsmReset();
		END_IF

		ASMR_INTERNAL_ERROR:

	END_CASE

	fbLogResetStep(); (* log state machine *)

END_PROGRAM
```

#### Init.st - Init code
```iecst
PROGRAM _INIT
	gSegA1;gSegA2;gSegA3;gSegA4;gSegA5;gSegA6;gSegA7;gSegA8;gSegA9;gSegA10;gSegA11;gSegA12;gSegA13;gSegA14;
	gSegB1;gSegB2;gSegB3;gSegB4;gSegB5;gSegB6;gSegB7;gSegB8;gSegB9;gSegB10;gSegB11;gSegB12;gSegB13;gSegB14;gSegB15;gSegB16;gSegB17;gSegB18;
	gSecOvalA;
	gSecOvalB;
	gSecB7;

	pDefectSegment := ADR(gSegB7);

	fbReadStatus.Assembly := ADR(gAssembly_1);
	fbReadStatus.Enable := TRUE;

	fbReadInfo.Assembly := fbReadStatus.Assembly;
	fbReadInfo.Enable := TRUE;

	fbGetInfo.Assembly := fbReadStatus.Assembly;

	fbPowerOn.Assembly := fbReadStatus.Assembly;

	fbPowerOff.Assembly := fbReadStatus.Assembly;

	fbStartShuttles.Sector := gSecCompleteLoop1;
	fbStartShuttles.TargetSector := gSecCompleteLoop1;
	fbStartShuttles.Acceleration := 4.0;
	fbStartShuttles.Deceleration := 4.0;
	fbStartShuttles.Velocity := 2.0;
	fbStartShuttles.Jerk := 0.0;
	fbStartShuttles.Direction := mcDIR_POSITIVE;

	fbAddSimShuttle.Sector := ADR(gSecCompleteLoop1);
	fbAddSimShuttle.Position := 0.5;

	fbAddSimShuttle.AdvancedParameters.Velocity := 0.0;
	fbAddSimShuttle.AdvancedParameters.Orientation := mcDIR_POSITIVE;
	fbAddSimShuttle.AdvancedParameters.Deceleration := 6.0;
	fbAddSimShuttle.AdvancedParameters.Virtual := FALSE;

	fbCatchShuttle.ProcessPoint := PP_ErrorPosition1;
	fbCatchShuttle.Enable := TRUE;

	fbAsmReset.Assembly := ADR(gAssembly_1);

	fbRecorder.AssemblyName := 'gAssembly_1';
	fbRecorder.FileDeviceName := 'Diagnosis';
	fbRecorder.FileNamePrefix := 'Demo_';
	fbRecorder.MaxNumberOfRecordings := 10;
	fbRecorder.DataAddress := ADR(shuttleData);
	fbRecorder.DataSize := SIZEOF(shuttleData); (* type of McAcpTrakShuttleData[] if no shuttle user data is defined, see MC_BR_AsmCopyShuttleData_AcpTrak *)
	fbRecorder.UserDataSize := 0;
	fbRecorder.Enable := TRUE;

	fbWebServices.AssemblyName := fbRecorder.AssemblyName;
	fbWebServices.DataAddress := fbRecorder.DataAddress;
	fbWebServices.DataSize := fbRecorder.DataSize;
	fbWebServices.UserDataSize := fbRecorder.UserDataSize;
	fbWebServices.Enable := TRUE;

	assemblyCtrl.Para.NumberOfSimulatedShuttles := 10;
	assemblyCtrl.SizeOf := SIZEOF(assemblyCtrl);

	step := ASM_INIT;

	fbLogStep( Enable := FALSE, LogName := 'MyTrak', SignalName := 'AssCtrl1 Step', EventID := TRAK_BASIC_INFO_ID );
	fbLogStep.Enable := TRUE;

	fbLogResetStep( Enable := FALSE, LogName := 'MyTrak', SignalName := 'AssCtrl1 ResetStep', EventID := TRAK_BASIC_INFO_ID );
	fbLogResetStep.Enable := TRUE;
END_PROGRAM
```

#### Variables.var - Local variables
```iecst
VAR
	fbStartShuttles : TL_StartShuttlesInSector;
	fbLogResetStep : TD_LogWatchSTRING;
	fbLogStep : TD_LogWatchSTRING;
	fbAddSimShuttle : MC_BR_SecAddShuttle_AcpTrak;
	fbPowerOff : MC_BR_AsmPowerOff_AcpTrak;
	fbPowerOn : MC_BR_AsmPowerOn_AcpTrak;
	fbGetInfo : MC_BR_AsmGetInfo_AcpTrak;
	fbReadInfo : MC_BR_AsmReadInfo_AcpTrak;
	fbReadStatus : MC_BR_AsmReadStatus_AcpTrak;
	fbWebServices : TD_WebServices;
	fbCatchShuttle : TL_CatchShuttle;
	pDefectSegment : {REDUND_UNREPLICABLE} UDINT;
	fbRecorder : TD_Recorder;
	step : AssemblyStepEnum;
	fbAsmReset : MC_BR_AsmReset_AcpTrak;
	fbSegCommandError : TD_SegCommandError;
	assemblyCtrl : AssemblyType;
	shuttleData : ARRAY[0..49] OF McAcpTrakShuttleData;
	shuttleCounter : DINT;
END_VAR
```

### Program Logical/Trak/AssCtrl2 (IEC)

- Cyclic.st (reference to Logical/Trak/AssCtrl1/Cyclic.st)

#### Init.st - Init code
```iecst
PROGRAM _INIT
	gSegC1;gSegC2;gSegC3;gSegC4;gSegC5;gSegC6;gSegC7;gSegC8;gSegC9;gSegC10;gSegC11;gSegC12;
	gSecC1;

	pDefectSegment := ADR(gSegC7);

	fbReadStatus.Assembly := ADR(gAssembly_2);
	fbReadStatus.Enable := TRUE;

	fbReadInfo.Assembly := fbReadStatus.Assembly;
	fbReadInfo.Enable := TRUE;

	fbGetInfo.Assembly := fbReadStatus.Assembly;

	fbPowerOn.Assembly := fbReadStatus.Assembly;

	fbPowerOff.Assembly := fbReadStatus.Assembly;

	fbStartShuttles.Sector := gSecOvalC;
	fbStartShuttles.TargetSector := gSecOvalC;
	fbStartShuttles.Acceleration := 4.0;
	fbStartShuttles.Deceleration := 4.0;
	fbStartShuttles.Velocity := 2.0;
	fbStartShuttles.Jerk := 0.0;
	fbStartShuttles.Direction := mcDIR_POSITIVE;

	fbAddSimShuttle.Sector := ADR(gSecOvalC);
	fbAddSimShuttle.Position := 0.5;

	fbAddSimShuttle.AdvancedParameters.Velocity := 0.0;
	fbAddSimShuttle.Orientation := mcDIR_POSITIVE;
	fbAddSimShuttle.AdvancedParameters.Deceleration := 6.0;
	fbAddSimShuttle.AdvancedParameters.Virtual := FALSE;

	fbCatchShuttle.ProcessPoint := PP_ErrorPosition2;
	fbCatchShuttle.Enable := TRUE;

	fbAsmReset.Assembly := ADR(gAssembly_2);

	fbRecorder.AssemblyName := 'gAssembly_2';
	fbRecorder.FileDeviceName := 'Diagnosis';
	fbRecorder.FileNamePrefix := 'Demo_';
	fbRecorder.MaxNumberOfRecordings := 10;
	fbRecorder.DataAddress := ADR(shuttleData);
	fbRecorder.DataSize := SIZEOF(shuttleData); (* type of McAcpTrakShuttleData[] if no shuttle user data is defined, see MC_BR_AsmCopyShuttleData_AcpTrak *)
	fbRecorder.UserDataSize := 0;
	fbRecorder.Enable := TRUE;

	fbWebServices.AssemblyName := fbRecorder.AssemblyName;
	fbWebServices.DataAddress := fbRecorder.DataAddress;
	fbWebServices.DataSize := fbRecorder.DataSize;
	fbWebServices.UserDataSize := fbRecorder.UserDataSize;
	fbWebServices.Enable := TRUE;

	assemblyCtrl.Para.NumberOfSimulatedShuttles := 10;
	assemblyCtrl.SizeOf := SIZEOF(assemblyCtrl);

	step := ASM_INIT;

	fbLogStep( Enable := FALSE, LogName := 'MyTrak', SignalName := 'AssCtrl2 Step', EventID := TRAK_BASIC_INFO_ID );
	fbLogStep.Enable := TRUE;

	fbLogResetStep( Enable := FALSE, LogName := 'MyTrak', SignalName := 'AssCtrl2 ResetStep', EventID := TRAK_BASIC_INFO_ID );
	fbLogResetStep.Enable := TRUE;

END_PROGRAM
```

- Variables.var (reference to Logical/Trak/AssCtrl1/Variables.var)

#### Variables.var - not listed in the package file held
```iecst
VAR
	fbStartShuttles : TL_StartShuttlesInSector;
	fbLogResetStep : TD_LogWatchSTRING;
	fbLogStep : TD_LogWatchSTRING;
	fbAddSimShuttle : MC_BR_SecAddShuttle_AcpTrak;
	fbPowerOff : MC_BR_AsmPowerOff_AcpTrak;
	fbPowerOn : MC_BR_AsmPowerOn_AcpTrak;
	fbGetInfo : MC_BR_AsmGetInfo_AcpTrak;
	fbReadInfo : MC_BR_AsmReadInfo_AcpTrak;
	fbReadStatus : MC_BR_AsmReadStatus_AcpTrak;
	fbWebServices : TD_WebServices;
	pDefectSegment : {REDUND_UNREPLICABLE} UDINT;
	fbCatchShuttle : TL_CatchShuttle;
	fbRecorder : TD_Recorder;
	step : AssemblyStepEnum;
	fbAsmReset : MC_BR_AsmReset_AcpTrak;
	fbSegCommandError : TD_SegCommandError;
	assemblyCtrl : AssemblyType;
	shuttleData : ARRAY[0..49] OF McAcpTrakShuttleData;
	shuttleCounter : DINT;
END_VAR
```

### Program Logical/Trak/AssCtrl (IEC)
